# B&R Automation Studio project EFI (part 5)

### Hardware
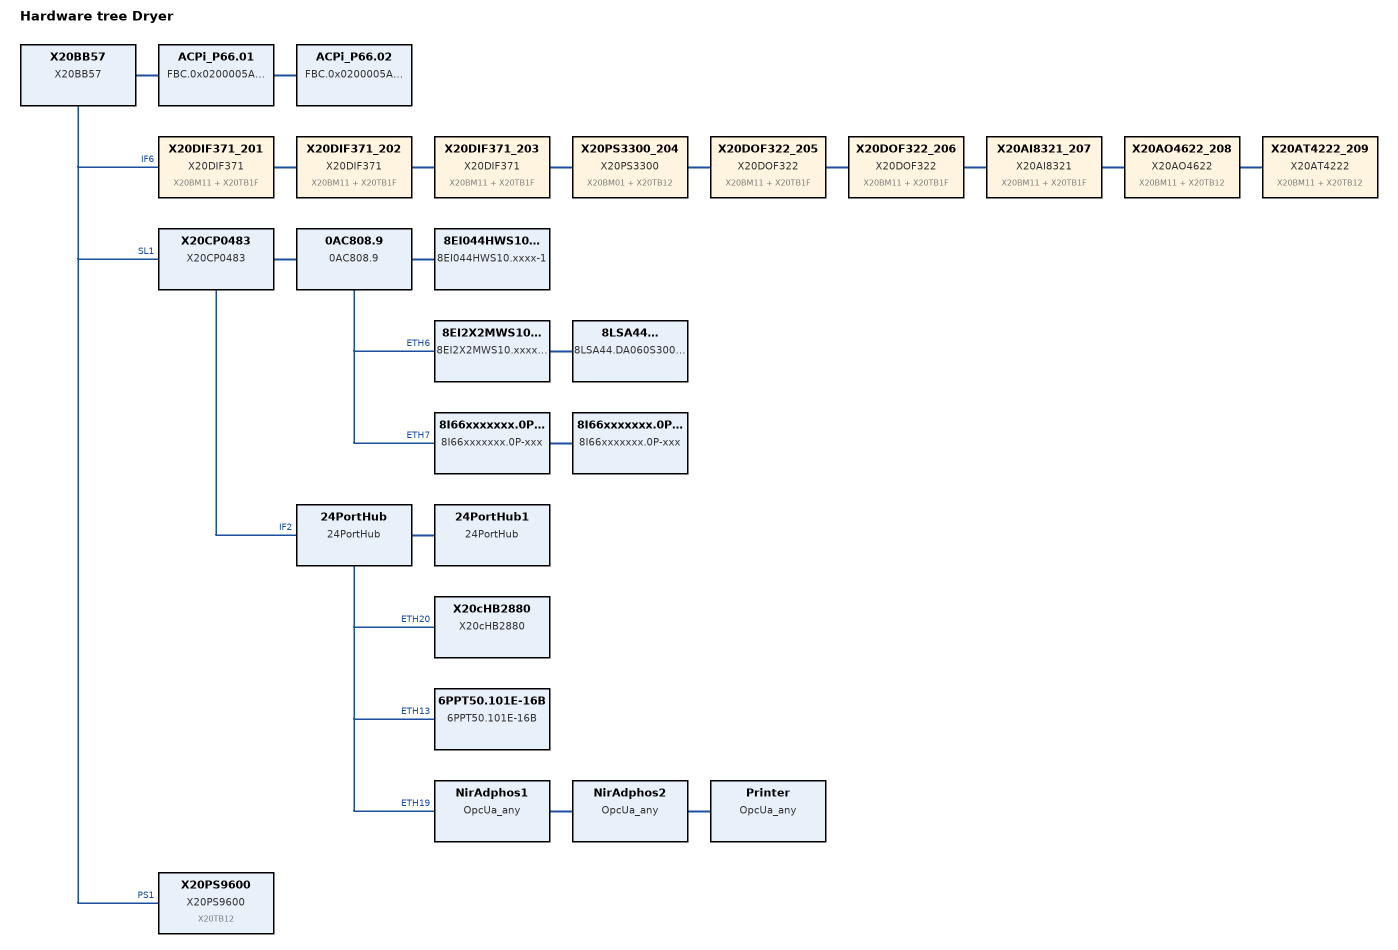
```
0AC808.9 : 0AC808.9 v1.0.0.0  [ETH1 -> X20CP0483.IF3 [Cable Type=PowerlinkCable, Length=10, Version=1.0.0.3]; ETH5 -> 8EI044HWS10.xxxx-1_BELT.PLK1 [Cable Type=PowerlinkCable, Length=10, Version=1.0.0.3]; ETH6 -> 8EI2X2MWS10.xxxx-1.PLK1 [Cable Type=PowerlinkCable, Length=10, Version=1.0.0.3]; ETH7 -> 8I66xxxxxxx.0P-81.PLK1 [Cable Type=PowerlinkCable, Length=10, Version=1.0.0.3]]
24PortHub : 24PortHub v1.0.0.1  [ETH7 -> X20CP0483.IF2 [Cable Type=PowerlinkCable, Length=10, Version=1.0.0.3]; ETH13 -> 6PPT50.101E-16B.ETH1 [Cable Type=PowerlinkCable, Length=10, Version=1.0.0.3]; ETH19 -> NirAdphos1.ETH1 [Cable Type=PowerlinkCable, Length=10, Version=1.0.0.3]; ETH20 -> X20cHB2880.ETH1 [Cable Type=PowerlinkCable, Length=10, Version=1.0.0.3]; ETH24 -> 24PortHub1.ETH3 [Cable Type=PowerlinkCable, Length=10, Version=1.0.0.3]]
24PortHub1 : 24PortHub v1.0.0.1  [ETH3 -> 24PortHub.ETH24 [Cable Type=PowerlinkCable, Length=10, Version=1.0.0.3]]
6PPT50.101E-16B : 6PPT50.101E-16B v1.3.8.0  [ETH1 -> 24PortHub.ETH13 [Cable Type=PowerlinkCable, Length=10, Version=1.0.0.3]]
  Terminal = true
  Startmode = 2
  ShowBootlogoWeb = 1
  Mode = Manual
  InternetAddress = 192.168.125.48
  Subnetmask = 255.255.255.0
  Hostname = efi_dryer_hmi
  Screensaver = 1
  Screensavertype = 0
  ActivateBuzzer = 1
  PasswordVNC = 
  SelectedFavoriteWeb = 192.168.125.47:81/index.html
  Favorites_Web1 = 
  BrowserVKeyboard = 0
  PasswordCIFS = 
  PasswordService = 
  ANSLAuthUserName = 
8EI044HWS10.xxxx-1_BELT : 8EI044HWS10.xxxx-1 v2.3.1.1  [PLK1 -> 0AC808.9.ETH5 [Cable Type=PowerlinkCable, Length=10, Version=1.0.0.3]]
  MotionTP = Acp10Arnc0
  Ax1Interface = Ax1EnDat
8EI2X2MWS10.xxxx-1 : 8EI2X2MWS10.xxxx-1 v2.3.1.1  [PLK1 -> 0AC808.9.ETH6 (NodeNumber=21) [Cable Type=PowerlinkCable, Length=10, Version=1.0.0.3]; EC1 -> 8LSA44.DA060S300-3.EC]
  MotionTP = Acp10Arnc0
  Ax1Interface = Ax1EnDat
8I66xxxxxxx.0P-81 : 8I66xxxxxxx.0P-xxx v2.5.1.0  [PLK1 -> 0AC808.9.ETH7 (NodeNumber=81) [Cable Type=PowerlinkCable, Length=10, Version=1.0.0.3]; PLK2 -> 8I66xxxxxxx.0P-82.PLK1 (NodeNumber=81) [Cable Type=PowerlinkCable, Length=10, Version=1.0.0.3]]
  FunctionModel = Standard
  Supervision = off
  UnitOfSetpoint = Rpm
  IOM_AIDP1 = LFT
  IOM_AIDP2 = LCR
  IOM_AIDP3 = OTRN
  IOM_AIDP4 = IL1R
  IOM_AIDP5 = AI1R
  IOM_AIDP6 = AI2R
  IOM_AIDP7 = AI3R
  IOM_AIDP8 = OL1I
  IOM_AIDP9 = AO1I
  IOM_R1ctrl = mapped
  IOM_R2ctrl = mapped
  IOM_LO1ctrl = mapped
  IOM_AO1ctrl = mapped
  Sel_AO1T = 0A
  Sel_NameplateMask = 8Ix6T401500_IEC
  Cfg_NSP = 2940
  Cfg_NCR = 277
  Cfg_COS = 82
  Sel_TUN = AUTO
8I66xxxxxxx.0P-82 : 8I66xxxxxxx.0P-xxx v2.5.1.0  [PLK1 -> 8I66xxxxxxx.0P-81.PLK2 [Cable Type=PowerlinkCable, Length=10, Version=1.0.0.3]]
  FunctionModel = Standard
  Supervision = off
  UnitOfSetpoint = Rpm
  IOM_AIDP1 = LFT
  IOM_AIDP2 = LCR
  IOM_AIDP3 = OTRN
  IOM_AIDP4 = IL1R
  IOM_AIDP5 = AI1R
  IOM_AIDP6 = AI2R
  IOM_AIDP7 = AI3R
  IOM_AIDP8 = OL1I
  IOM_AIDP9 = AO1I
  IOM_R1ctrl = mapped
  IOM_R2ctrl = mapped
  IOM_LO1ctrl = mapped
  IOM_AO1ctrl = mapped
  Sel_AO1T = 0A
  Sel_NameplateMask = 8Ix6T401500_IEC
  Cfg_NSP = 2940
  Cfg_NCR = 277
  Cfg_COS = 82
  Sel_TUN = AUTO
8LSA44.DA060S300-3 : 8LSA44.DA060S300-3 v1.0.10.37  [EC -> 8EI2X2MWS10.xxxx-1.EC1; MT -> 8EI2X2MWS10.xxxx-1.MT1]
ACPi_P66.01 : FBC.0x0200005A.320.ACPi_P66_P76 v1.3 (OrderNumber=ACPi_P66_P76)  [CAN1 -> X20BB57.IF7 (NodeNumber=81)]
  p2002sub5_connecttomaster = 2
  p2016sub3_connecttomaster = 1
  p2016subd_connecttomaster = 5
  p2016sub21_connecttomaster = 1
  p2016sub22_connecttomaster = 1
  p2016sub3e_connecttomaster = 5
  p2029sub16_connecttomaster = 2
  p2038sub2_connecttomaster = 4
  p2038sub3_connecttomaster = 4
  p2038sub4_connecttomaster = 2
  p2038sub5_connecttomaster = 2
  p203csub2_connecttomaster = 5
  p203csub3_connecttomaster = 5
  p6040_connecttomaster = 0
  p6041_connecttomaster = 0
  p6042_connecttomaster = 0
  p6044_connecttomaster = 0
  p6077_connecttomaster = 1
  p1800_transmissionselection = 2
  p1801_transmissionselection = 2
  p1802_transmissionselection = 2
ACPi_P66.02 : FBC.0x0200005A.320.ACPi_P66_P76 v1.3 (OrderNumber=ACPi_P66_P76)  [CAN1 -> ACPi_P66.01.CAN2]
  p2002sub5_connecttomaster = 2
  p2016sub3_connecttomaster = 1
  p2016subd_connecttomaster = 5
  p2016sub21_connecttomaster = 1
  p2016sub22_connecttomaster = 1
  p2016sub3e_connecttomaster = 5
  p2029sub16_connecttomaster = 2
  p2038sub2_connecttomaster = 4
  p2038sub3_connecttomaster = 4
  p2038sub4_connecttomaster = 2
  p2038sub5_connecttomaster = 2
  p203csub2_connecttomaster = 5
  p203csub3_connecttomaster = 5
  p6040_connecttomaster = 0
  p6041_connecttomaster = 0
  p6042_connecttomaster = 0
  p6044_connecttomaster = 0
  p6077_connecttomaster = 1
  p1800_transmissionselection = 2
  p1801_transmissionselection = 2
  p1802_transmissionselection = 2
NirAdphos1 : OpcUa_any v1.0.0.1  [ETH1 -> 24PortHub.ETH19 [Cable Type=PowerlinkCable, Length=10, Version=1.0.0.3]; ETH2 -> NirAdphos2.ETH1 [Cable Type=PowerlinkCable, Length=10, Version=1.0.0.3]]
  ServerDiagnostics = on
  ServerEndpointUrl = opc.tcp://192.168.125.91:4840
  PnPTimeout = 2500
  SecurityMsgMode = 0
  Channel1
  ChannelID1 = HMI
  ChannelBrowsePath1 = /0:Root/0:Objects/3:ServerInterfaces/4:SendData/4:DB11_HMI_out/4:HMI
  ChannelType1 = INT
  Channel2
  ChannelID2 = Hardware
  ChannelBrowsePath2 = /0:Root/0:Objects/3:ServerInterfaces/4:SendData/4:DB11_HMI_out/4:Hardware
  ChannelType2 = INT
  Channel3
  ChannelID3 = Software
  ChannelBrowsePath3 = /0:Root/0:Objects/3:ServerInterfaces/4:SendData/4:DB11_HMI_out/4:Software
  ChannelType3 = INT
  Channel4
  ChannelID4 = Interface
  ChannelBrowsePath4 = /0:Root/0:Objects/3:ServerInterfaces/4:SendData/4:DB11_HMI_out/4:interface
  ChannelType4 = INT
  Channel5
  ChannelID5 = NIRno
  ChannelBrowsePath5 = /0:Root/0:Objects/3:ServerInterfaces/4:SendData/4:DB11_HMI_out/4:general/4:NIRno
  ChannelType5 = INT
  Channel6
  ChannelID6 = NIRwidth
  ChannelBrowsePath6 = /0:Root/0:Objects/3:ServerInterfaces/4:SendData/4:DB11_HMI_out/4:general/4:NIRwidth
  ChannelType6 = INT
  Channel7
  ChannelID7 = calPower
  ChannelBrowsePath7 = /0:Root/0:Objects/3:ServerInterfaces/4:SendData/4:DB11_HMI_out/4:general/4:calPower
  ChannelType7 = INT
  Channel8
  ChannelID8 = speed
  ChannelBrowsePath8 = /0:Root/0:Objects/3:ServerInterfaces/4:SendData/4:DB11_HMI_out/4:general/4:speed
  ChannelType8 = REAL
  Channel9
  ChannelID9 = Watchdog1
  ChannelBrowsePath9 = /0:Root/0:Objects/3:ServerInterfaces/4:SendData/4:DB11_HMI_out/4:general/4:Watchdog
  Channel10
  ChannelID10 = EmFailNo_1
  ChannelBrowsePath10 = /0:Root/0:Objects/3:ServerInterfaces/4:SendData/4:DB11_HMI_out/4:module/4:[1]/4:EmFailNo
  ChannelType10 = USINT
  Channel11
  ChannelID11 = EmFailNo_2
  ChannelBrowsePath11 = /0:Root/0:Objects/3:ServerInterfaces/4:SendData/4:DB11_HMI_out/4:module/4:[2]/4:EmFailNo
  ChannelType11 = USINT
  Channel12
  ChannelID12 = ExhAirRunning_1
  ChannelBrowsePath12 = /0:Root/0:Objects/3:ServerInterfaces/4:SendData/4:DB11_HMI_out/4:module/4:[1]/4:ExhAirRunning
  Channel13
  ChannelID13 = ExhAirRunning_2
  ChannelBrowsePath13 = /0:Root/0:Objects/3:ServerInterfaces/4:SendData/4:DB11_HMI_out/4:module/4:[2]/4:ExhAirRunning
  Channel14
  ChannelID14 = NIRstatus_1
  ChannelBrowsePath14 = /0:Root/0:Objects/3:ServerInterfaces/4:SendData/4:DB11_HMI_out/4:module/4:[1]/4:NIRstatus
  ChannelType14 = INT
  Channel15
  ChannelID15 = NIRstatus_2
  ChannelBrowsePath15 = /0:Root/0:Objects/3:ServerInterfaces/4:SendData/4:DB11_HMI_out/4:module/4:[2]/4:NIRstatus
  ChannelType15 = INT
  Channel16
  ChannelID16 = airPressIn_1
  ChannelBrowsePath16 = /0:Root/0:Objects/3:ServerInterfaces/4:SendData/4:DB11_HMI_out/4:module/4:[1]/4:airPressIn
  ChannelType16 = REAL
  Channel17
  ChannelID17 = airPressIn_2
  ChannelBrowsePath17 = /0:Root/0:Objects/3:ServerInterfaces/4:SendData/4:DB11_HMI_out/4:module/4:[2]/4:airPressIn
  ChannelType17 = REAL
  Channel18
  ChannelID18 = airPressOut_1
  ChannelBrowsePath18 = /0:Root/0:Objects/3:ServerInterfaces/4:SendData/4:DB11_HMI_out/4:module/4:[1]/4:airPressOut
  ChannelType18 = REAL
  Channel19
  ChannelID19 = airPressOut_2
  ChannelBrowsePath19 = /0:Root/0:Objects/3:ServerInterfaces/4:SendData/4:DB11_HMI_out/4:module/4:[2]/4:airPressOut
  ChannelType19 = REAL
  Channel20
  ChannelID20 = airFilter_1
  ChannelBrowsePath20 = /0:Root/0:Objects/3:ServerInterfaces/4:SendData/4:DB11_HMI_out/4:module/4:[1]/4:airFilter
  ChannelType20 = INT
  Channel21
  ChannelID21 = airFilter_2
  ChannelBrowsePath21 = /0:Root/0:Objects/3:ServerInterfaces/4:SendData/4:DB11_HMI_out/4:module/4:[2]/4:airFilter
  ChannelType21 = INT
  Channel22
  ChannelID22 = actSpeedIn_1
  ChannelBrowsePath22 = /0:Root/0:Objects/3:ServerInterfaces/4:SendData/4:DB11_HMI_out/4:module/4:[1]/4:actSpeedIn
  ChannelType22 = INT
  Channel23
  ChannelID23 = actSpeedIn_2
  ChannelBrowsePath23 = /0:Root/0:Objects/3:ServerInterfaces/4:SendData/4:DB11_HMI_out/4:module/4:[2]/4:actSpeedIn
  ChannelType23 = INT
  Channel24
  ChannelID24 = actSpeedOut_1
  ChannelBrowsePath24 = /0:Root/0:Objects/3:ServerInterfaces/4:SendData/4:DB11_HMI_out/4:module/4:[1]/4:actSpeedOut
  ChannelType24 = INT
  Channel25
  ChannelID25 = actSpeedOut_2
  ChannelBrowsePath25 = /0:Root/0:Objects/3:ServerInterfaces/4:SendData/4:DB11_HMI_out/4:module/4:[2]/4:actSpeedOut
  ChannelType25 = INT
  Channel26
  ChannelID26 = actPower_1
  ChannelBrowsePath26 = /0:Root/0:Objects/3:ServerInterfaces/4:SendData/4:DB11_HMI_out/4:module/4:[1]/4:actPower
  ChannelType26 = INT
  Channel27
  ChannelID27 = actPower_2
  ChannelBrowsePath27 = /0:Root/0:Objects/3:ServerInterfaces/4:SendData/4:DB11_HMI_out/4:module/4:[2]/4:actPower
  ChannelType27 = INT
  Channel28
  ChannelID28 = Watchdog2
  ChannelBrowsePath28 = /0:Root/0:Objects/3:ServerInterfaces/4:SendData/4:DB11_HMI_out/4:general/4:Watchdog
  Channel29
  ChannelID29 = Reset
  ChannelBrowsePath29 = /0:Root/0:Objects/3:ServerInterfaces/5:RecData/5:DB10_HMI_in/5:reset
  ChannelDirection29 = OUT
  Channel30
  ChannelID30 = Pend
  ChannelBrowsePath30 = /0:Root/0:Objects/3:ServerInterfaces/5:RecData/5:DB10_HMI_in/5:product/5:Pend
  ChannelDirection30 = OUT
  ChannelType30 = REAL
  Channel31
  ChannelID31 = Pstart
  ChannelBrowsePath31 = /0:Root/0:Objects/3:ServerInterfaces/5:RecData/5:DB10_HMI_in/5:product/5:Pstart
  ChannelDirection31 = OUT
  ChannelType31 = REAL
  Channel32
  ChannelID32 = Vend
  ChannelBrowsePath32 = /0:Root/0:Objects/3:ServerInterfaces/5:RecData/5:DB10_HMI_in/5:product/5:Vend
  ChannelDirection32 = OUT
  ChannelType32 = REAL
  Channel33
  ChannelID33 = Vstart
  ChannelBrowsePath33 = /0:Root/0:Objects/3:ServerInterfaces/5:RecData/5:DB10_HMI_in/5:product/5:Vstart
  ChannelDirection33 = OUT
  ChannelType33 = REAL
  Channel34
  ChannelID34 = AdjPos
  ChannelBrowsePath34 = /0:Root/0:Objects/3:ServerInterfaces/5:RecData/5:DB10_HMI_in/5:product/5:adjPos
  ChannelDirection34 = OUT
  ChannelType34 = INT
  Channel35
  ChannelID35 = WebWidth
  ChannelBrowsePath35 = /0:Root/0:Objects/3:ServerInterfaces/5:RecData/5:DB10_HMI_in/5:product/5:webWidth
  ChannelDirection35 = OUT
  ChannelType35 = INT
  Channel36
  ChannelID36 = Adjust_1
  ChannelBrowsePath36 = /0:Root/0:Objects/3:ServerInterfaces/5:RecData/5:DB10_HMI_in/5:module/5:[1]/5:adjust
  ChannelDirection36 = OUT
  ChannelType36 = INT
  Channel37
  ChannelID37 = Adjust_2
  ChannelBrowsePath37 = /0:Root/0:Objects/3:ServerInterfaces/5:RecData/5:DB10_HMI_in/5:module/5:[2]/5:adjust
  ChannelDirection37 = OUT
  ChannelType37 = INT
  Channel38
  ChannelID38 = EnableMod_1
  ChannelBrowsePath38 = /0:Root/0:Objects/3:ServerInterfaces/5:RecData/5:DB10_HMI_in/5:module/5:[1]/5:enableMod
  ChannelDirection38 = OUT
  Channel39
  ChannelID39 = EnableMod_2
  ChannelBrowsePath39 = /0:Root/0:Objects/3:ServerInterfaces/5:RecData/5:DB10_HMI_in/5:module/5:[2]/5:enableMod
  ChannelDirection39 = OUT
  Channel40
  ChannelID40 = WatchdogOut
  ChannelBrowsePath40 = /0:Root/0:Objects/3:ServerInterfaces/5:RecData/5:DB10_HMI_in/5:Watchdog
  ChannelDirection40 = OUT
  Channel41
  ChannelID41 = Enable_DDC
  ChannelBrowsePath41 = /0:Root/0:Objects/3:ServerInterfaces/5:RecData/5:DB10_HMI_in/5:DDCon
  ChannelDirection41 = OUT
  Channel42
  ChannelID42 = NIR1_Int1
  ChannelBrowsePath42 = /0:Root/0:Objects/3:ServerInterfaces/5:RecData/5:DB10_HMI_in/5:intensity/5:intensity/5:[1]
  ChannelDirection42 = OUT
  ChannelType42 = INT
  Channel43
  ChannelID43 = NIR1_Int2
  ChannelBrowsePath43 = /0:Root/0:Objects/3:ServerInterfaces/5:RecData/5:DB10_HMI_in/5:intensity/5:intensity/5:[2]
  ChannelDirection43 = OUT
  ChannelType43 = INT
  Channel44
  ChannelID44 = NIR1_Int3
  ChannelBrowsePath44 = /0:Root/0:Objects/3:ServerInterfaces/5:RecData/5:DB10_HMI_in/5:intensity/5:intensity/5:[3]
  ChannelDirection44 = OUT
  ChannelType44 = INT
  Channel45
  ChannelID45 = NIR1_Int4
  ChannelBrowsePath45 = /0:Root/0:Objects/3:ServerInterfaces/5:RecData/5:DB10_HMI_in/5:intensity/5:intensity/5:[4]
  ChannelDirection45 = OUT
  ChannelType45 = INT
  Channel46
  ChannelID46 = NIR1_Int5
  ChannelBrowsePath46 = /0:Root/0:Objects/3:ServerInterfaces/5:RecData/5:DB10_HMI_in/5:intensity/5:intensity/5:[5]
  ChannelDirection46 = OUT
  ChannelType46 = INT
  Channel47
  ChannelID47 = NIR1_Int6
  ChannelBrowsePath47 = /0:Root/0:Objects/3:ServerInterfaces/5:RecData/5:DB10_HMI_in/5:intensity/5:intensity/5:[6]
  ChannelDirection47 = OUT
  ChannelType47 = INT
  Channel48
  ChannelID48 = NIR1_Int7
  ChannelBrowsePath48 = /0:Root/0:Objects/3:ServerInterfaces/5:RecData/5:DB10_HMI_in/5:intensity/5:intensity/5:[7]
  ChannelDirection48 = OUT
  ChannelType48 = INT
  Channel49
  ChannelID49 = NIR1_Int8
  ChannelBrowsePath49 = /0:Root/0:Objects/3:ServerInterfaces/5:RecData/5:DB10_HMI_in/5:intensity/5:intensity/5:[8]
  ChannelDirection49 = OUT
  ChannelType49 = INT
  Channel50
  ChannelID50 = NIR1_Int9
  ChannelBrowsePath50 = /0:Root/0:Objects/3:ServerInterfaces/5:RecData/5:DB10_HMI_in/5:intensity/5:intensity/5:[9]
  ChannelDirection50 = OUT
  ChannelType50 = INT
  Channel51
  ChannelID51 = NIR1_Int10
  ChannelBrowsePath51 = /0:Root/0:Objects/3:ServerInterfaces/5:RecData/5:DB10_HMI_in/5:intensity/5:intensity/5:[10]
  ChannelDirection51 = OUT
  ChannelType51 = INT
  Channel52
  ChannelID52 = NIR1_Int11
  ChannelBrowsePath52 = /0:Root/0:Objects/3:ServerInterfaces/5:RecData/5:DB10_HMI_in/5:intensity/5:intensity/5:[11]
  ChannelDirection52 = OUT
  ChannelType52 = INT
  Channel53
  ChannelID53 = NIR1_Int12
  ChannelBrowsePath53 = /0:Root/0:Objects/3:ServerInterfaces/5:RecData/5:DB10_HMI_in/5:intensity/5:intensity/5:[12]
  ChannelDirection53 = OUT
  ChannelType53 = INT
  Channel54
  ChannelID54 = NIR1_Int13
  ChannelBrowsePath54 = /0:Root/0:Objects/3:ServerInterfaces/5:RecData/5:DB10_HMI_in/5:intensity/5:intensity/5:[13]
  ChannelDirection54 = OUT
  ChannelType54 = INT
  Channel55
  ChannelID55 = NIR1_Int14
  ChannelBrowsePath55 = /0:Root/0:Objects/3:ServerInterfaces/5:RecData/5:DB10_HMI_in/5:intensity/5:intensity/5:[14]
  ChannelDirection55 = OUT
  ChannelType55 = INT
  Channel56
  ChannelID56 = NIR1_Int15
  ChannelBrowsePath56 = /0:Root/0:Objects/3:ServerInterfaces/5:RecData/5:DB10_HMI_in/5:intensity/5:intensity/5:[15]
  ChannelDirection56 = OUT
  ChannelType56 = INT
  Channel57
  ChannelID57 = NIR1_Int16
  ChannelBrowsePath57 = /0:Root/0:Objects/3:ServerInterfaces/5:RecData/5:DB10_HMI_in/5:intensity/5:intensity/5:[16]
  ChannelDirection57 = OUT
  ChannelType57 = INT
  Channel58
  ChannelID58 = NIR1_Int17
  ChannelBrowsePath58 = /0:Root/0:Objects/3:ServerInterfaces/5:RecData/5:DB10_HMI_in/5:intensity/5:intensity/5:[17]
  ChannelDirection58 = OUT
  ChannelType58 = INT
  Channel59
  ChannelID59 = NIR1_Int18
  ChannelBrowsePath59 = /0:Root/0:Objects/3:ServerInterfaces/5:RecData/5:DB10_HMI_in/5:intensity/5:intensity/5:[18]
  ChannelDirection59 = OUT
  ChannelType59 = INT
  Channel60
  ChannelID60 = NIR1_Int19
  ChannelBrowsePath60 = /0:Root/0:Objects/3:ServerInterfaces/5:RecData/5:DB10_HMI_in/5:intensity/5:intensity/5:[19]
  ChannelDirection60 = OUT
  ChannelType60 = INT
  Channel61
  ChannelID61 = NIR1_Int20
  ChannelBrowsePath61 = /0:Root/0:Objects/3:ServerInterfaces/5:RecData/5:DB10_HMI_in/5:intensity/5:intensity/5:[20]
  ChannelDirection61 = OUT
  ChannelType61 = INT
  Channel62
  ChannelID62 = NIR1_Int21
  ChannelBrowsePath62 = /0:Root/0:Objects/3:ServerInterfaces/5:RecData/5:DB10_HMI_in/5:intensity/5:intensity/5:[21]
  ChannelDirection62 = OUT
  ChannelType62 = INT
  Channel63
  ChannelID63 = NIR1_Int22
  ChannelBrowsePath63 = /0:Root/0:Objects/3:ServerInterfaces/5:RecData/5:DB10_HMI_in/5:intensity/5:intensity/5:[22]
  ChannelDirection63 = OUT
  ChannelType63 = INT
  Channel64
  ChannelID64 = NIR1_Int23
  ChannelBrowsePath64 = /0:Root/0:Objects/3:ServerInterfaces/5:RecData/5:DB10_HMI_in/5:intensity/5:intensity/5:[23]
  ChannelDirection64 = OUT
  ChannelType64 = INT
  Channel65
  ChannelID65 = NIR1_Int24
  ChannelBrowsePath65 = /0:Root/0:Objects/3:ServerInterfaces/5:RecData/5:DB10_HMI_in/5:intensity/5:intensity/5:[24]
  ChannelDirection65 = OUT
  ChannelType65 = INT
  Channel66
  ChannelID66 = NIR1_Int25
  ChannelBrowsePath66 = /0:Root/0:Objects/3:ServerInterfaces/5:RecData/5:DB10_HMI_in/5:intensity/5:intensity/5:[25]
  ChannelDirection66 = OUT
  ChannelType66 = INT
  Channel67
  ChannelID67 = NIR1_Int26
  ChannelBrowsePath67 = /0:Root/0:Objects/3:ServerInterfaces/5:RecData/5:DB10_HMI_in/5:intensity/5:intensity/5:[26]
  ChannelDirection67 = OUT
  ChannelType67 = INT
  Channel68
  ChannelID68 = NIR1_Int27
  ChannelBrowsePath68 = /0:Root/0:Objects/3:ServerInterfaces/5:RecData/5:DB10_HMI_in/5:intensity/5:intensity/5:[27]
  ChannelDirection68 = OUT
  ChannelType68 = INT
  Channel69
  ChannelID69 = NIR1_Int28
  ChannelBrowsePath69 = /0:Root/0:Objects/3:ServerInterfaces/5:RecData/5:DB10_HMI_in/5:intensity/5:intensity/5:[28]
  ChannelDirection69 = OUT
  ChannelType69 = INT
  Channel70
  ChannelID70 = NIR1_Int29
  ChannelBrowsePath70 = /0:Root/0:Objects/3:ServerInterfaces/5:RecData/5:DB10_HMI_in/5:intensity/5:intensity/5:[29]
  ChannelDirection70 = OUT
  ChannelType70 = INT
  Channel71
  ChannelID71 = NIR1_Int30
  ChannelBrowsePath71 = /0:Root/0:Objects/3:ServerInterfaces/5:RecData/5:DB10_HMI_in/5:intensity/5:intensity/5:[30]
  ChannelDirection71 = OUT
  ChannelType71 = INT
  Channel72
  ChannelID72 = NIR1_Int31
  ChannelBrowsePath72 = /0:Root/0:Objects/3:ServerInterfaces/5:RecData/5:DB10_HMI_in/5:intensity/5:intensity/5:[31]
  ChannelDirection72 = OUT
  ChannelType72 = INT
  Channel73
  ChannelID73 = NIR1_Int32
  ChannelBrowsePath73 = /0:Root/0:Objects/3:ServerInterfaces/5:RecData/5:DB10_HMI_in/5:intensity/5:intensity/5:[32]
  ChannelDirection73 = OUT
  ChannelType73 = INT
  Channel74
  ChannelID74 = NIR1_Int33
  ChannelBrowsePath74 = /0:Root/0:Objects/3:ServerInterfaces/5:RecData/5:DB10_HMI_in/5:intensity/5:intensity/5:[33]
  ChannelDirection74 = OUT
  ChannelType74 = INT
  Channel75
  ChannelID75 = NIR1_Int34
  ChannelBrowsePath75 = /0:Root/0:Objects/3:ServerInterfaces/5:RecData/5:DB10_HMI_in/5:intensity/5:intensity/5:[34]
  ChannelDirection75 = OUT
  ChannelType75 = INT
  Channel76
  ChannelID76 = NIR1_Int35
  ChannelBrowsePath76 = /0:Root/0:Objects/3:ServerInterfaces/5:RecData/5:DB10_HMI_in/5:intensity/5:intensity/5:[35]
  ChannelDirection76 = OUT
  ChannelType76 = INT
  Channel77
  ChannelID77 = NIR1_Int36
  ChannelBrowsePath77 = /0:Root/0:Objects/3:ServerInterfaces/5:RecData/5:DB10_HMI_in/5:intensity/5:intensity/5:[36]
  ChannelDirection77 = OUT
  ChannelType77 = INT
  Channel78
  ChannelID78 = NIR1_Int37
  ChannelBrowsePath78 = /0:Root/0:Objects/3:ServerInterfaces/5:RecData/5:DB10_HMI_in/5:intensity/5:intensity/5:[37]
  ChannelDirection78 = OUT
  ChannelType78 = INT
  Channel79
  ChannelID79 = NIR1_Int38
  ChannelBrowsePath79 = /0:Root/0:Objects/3:ServerInterfaces/5:RecData/5:DB10_HMI_in/5:intensity/5:intensity/5:[38]
  ChannelDirection79 = OUT
  ChannelType79 = INT
  Channel80
  ChannelID80 = NIR1_Int39
  ChannelBrowsePath80 = /0:Root/0:Objects/3:ServerInterfaces/5:RecData/5:DB10_HMI_in/5:intensity/5:intensity/5:[39]
  ChannelDirection80 = OUT
  ChannelType80 = INT
  Channel81
  ChannelID81 = NIR1_Int40
  ChannelBrowsePath81 = /0:Root/0:Objects/3:ServerInterfaces/5:RecData/5:DB10_HMI_in/5:intensity/5:intensity/5:[40]
  ChannelDirection81 = OUT
  ChannelType81 = INT
  Channel82
  ChannelID82 = NIR1_Int41
  ChannelBrowsePath82 = /0:Root/0:Objects/3:ServerInterfaces/5:RecData/5:DB10_HMI_in/5:intensity/5:intensity/5:[41]
  ChannelDirection82 = OUT
  ChannelType82 = INT
  Channel83
  ChannelID83 = NIR1_Int42
  ChannelBrowsePath83 = /0:Root/0:Objects/3:ServerInterfaces/5:RecData/5:DB10_HMI_in/5:intensity/5:intensity/5:[42]
  ChannelDirection83 = OUT
  ChannelType83 = INT
  Channel84
  ChannelID84 = NIR1_Int43
  ChannelBrowsePath84 = /0:Root/0:Objects/3:ServerInterfaces/5:RecData/5:DB10_HMI_in/5:intensity/5:intensity/5:[43]
  ChannelDirection84 = OUT
  ChannelType84 = INT
  Channel85
  ChannelID85 = NIR1_Int44
  ChannelBrowsePath85 = /0:Root/0:Objects/3:ServerInterfaces/5:RecData/5:DB10_HMI_in/5:intensity/5:intensity/5:[44]
  ChannelDirection85 = OUT
  ChannelType85 = INT
  Channel86
  ChannelID86 = NIR1_Int45
  ChannelBrowsePath86 = /0:Root/0:Objects/3:ServerInterfaces/5:RecData/5:DB10_HMI_in/5:intensity/5:intensity/5:[45]
  ChannelDirection86 = OUT
  ChannelType86 = INT
  Channel87
  ChannelID87 = NIR1_Int46
  ChannelBrowsePath87 = /0:Root/0:Objects/3:ServerInterfaces/5:RecData/5:DB10_HMI_in/5:intensity/5:intensity/5:[46]
  ChannelDirection87 = OUT
  ChannelType87 = INT
  Channel88
  ChannelID88 = NIR1_Int47
  ChannelBrowsePath88 = /0:Root/0:Objects/3:ServerInterfaces/5:RecData/5:DB10_HMI_in/5:intensity/5:intensity/5:[47]
  ChannelDirection88 = OUT
  ChannelType88 = INT
  Channel89
  ChannelID89 = NIR1_Int48
  ChannelBrowsePath89 = /0:Root/0:Objects/3:ServerInterfaces/5:RecData/5:DB10_HMI_in/5:intensity/5:intensity/5:[48]
  ChannelDirection89 = OUT
  ChannelType89 = INT
NirAdphos2 : OpcUa_any v1.0.0.1  [ETH1 -> NirAdphos1.ETH2 [Cable Type=PowerlinkCable, Length=10, Version=1.0.0.3]; ETH2 -> Printer.ETH1 [Cable Type=PowerlinkCable, Length=10, Version=1.0.0.3]]
  ServerDiagnostics = on
  ServerEndpointUrl = opc.tcp://192.168.125.92:4840
  PnPTimeout = 2500
  SecurityMsgMode = 0
  Channel1
  ChannelID1 = NIR2_Int1
  ChannelBrowsePath1 = /0:Root/0:Objects/3:ServerInterfaces/0:RecData/4:DB10_HMI_in/4:intensity/4:[1]
  ChannelDirection1 = OUT
  ChannelType1 = INT
  Channel2
  ChannelID2 = NIR2_Int2
  ChannelBrowsePath2 = /0:Root/0:Objects/3:ServerInterfaces/0:RecData/4:DB10_HMI_in/4:intensity/4:[2]
  ChannelDirection2 = OUT
  ChannelType2 = INT
  Channel3
  ChannelID3 = NIR2_Int3
  ChannelBrowsePath3 = /0:Root/0:Objects/3:ServerInterfaces/0:RecData/4:DB10_HMI_in/4:intensity/4:[3]
  ChannelDirection3 = OUT
  ChannelType3 = INT
  Channel4
  ChannelID4 = NIR2_Int4
  ChannelBrowsePath4 = /0:Root/0:Objects/3:ServerInterfaces/0:RecData/4:DB10_HMI_in/4:intensity/4:[4]
  ChannelDirection4 = OUT
  ChannelType4 = INT
  Channel5
  ChannelID5 = NIR2_Int5
  ChannelBrowsePath5 = /0:Root/0:Objects/3:ServerInterfaces/0:RecData/4:DB10_HMI_in/4:intensity/4:[5]
  ChannelDirection5 = OUT
  ChannelType5 = INT
  Channel6
  ChannelID6 = NIR2_Int6
  ChannelBrowsePath6 = /0:Root/0:Objects/3:ServerInterfaces/0:RecData/4:DB10_HMI_in/4:intensity/4:[6]
  ChannelDirection6 = OUT
  ChannelType6 = INT
  Channel7
  ChannelID7 = NIR2_Int7
  ChannelBrowsePath7 = /0:Root/0:Objects/3:ServerInterfaces/0:RecData/4:DB10_HMI_in/4:intensity/4:[7]
  ChannelDirection7 = OUT
  ChannelType7 = INT
  Channel8
  ChannelID8 = NIR2_Int8
  ChannelBrowsePath8 = /0:Root/0:Objects/3:ServerInterfaces/0:RecData/4:DB10_HMI_in/4:intensity/4:[8]
  ChannelDirection8 = OUT
  ChannelType8 = INT
  Channel9
  ChannelID9 = NIR2_Int9
  ChannelBrowsePath9 = /0:Root/0:Objects/3:ServerInterfaces/0:RecData/4:DB10_HMI_in/4:intensity/4:[9]
  ChannelDirection9 = OUT
  ChannelType9 = INT
  Channel10
  ChannelID10 = NIR2_Int10
  ChannelBrowsePath10 = /0:Root/0:Objects/3:ServerInterfaces/0:RecData/4:DB10_HMI_in/4:intensity/4:[10]
  ChannelDirection10 = OUT
  ChannelType10 = INT
  Channel11
  ChannelID11 = NIR2_Int11
  ChannelBrowsePath11 = /0:Root/0:Objects/3:ServerInterfaces/0:RecData/4:DB10_HMI_in/4:intensity/4:[11]
  ChannelDirection11 = OUT
  ChannelType11 = INT
  Channel12
  ChannelID12 = NIR2_Int12
  ChannelBrowsePath12 = /0:Root/0:Objects/3:ServerInterfaces/0:RecData/4:DB10_HMI_in/4:intensity/4:[12]
  ChannelDirection12 = OUT
  ChannelType12 = INT
  Channel13
  ChannelID13 = NIR2_Int13
  ChannelBrowsePath13 = /0:Root/0:Objects/3:ServerInterfaces/0:RecData/4:DB10_HMI_in/4:intensity/4:[13]
  ChannelDirection13 = OUT
  ChannelType13 = INT
  Channel14
  ChannelID14 = NIR2_Int14
  ChannelBrowsePath14 = /0:Root/0:Objects/3:ServerInterfaces/0:RecData/4:DB10_HMI_in/4:intensity/4:[14]
  ChannelDirection14 = OUT
  ChannelType14 = INT
  Channel15
  ChannelID15 = NIR2_Int15
  ChannelBrowsePath15 = /0:Root/0:Objects/3:ServerInterfaces/0:RecData/4:DB10_HMI_in/4:intensity/4:[15]
  ChannelDirection15 = OUT
  ChannelType15 = INT
  Channel16
  ChannelID16 = NIR2_Int16
  ChannelBrowsePath16 = /0:Root/0:Objects/3:ServerInterfaces/0:RecData/4:DB10_HMI_in/4:intensity/4:[16]
  ChannelDirection16 = OUT
  ChannelType16 = INT
  Channel17
  ChannelID17 = NIR2_Int17
  ChannelBrowsePath17 = /0:Root/0:Objects/3:ServerInterfaces/0:RecData/4:DB10_HMI_in/4:intensity/4:[17]
  ChannelDirection17 = OUT
  ChannelType17 = INT
  Channel18
  ChannelID18 = NIR2_Int18
  ChannelBrowsePath18 = /0:Root/0:Objects/3:ServerInterfaces/0:RecData/4:DB10_HMI_in/4:intensity/4:[18]
  ChannelDirection18 = OUT
  ChannelType18 = INT
  Channel19
  ChannelID19 = NIR2_Int19
  ChannelBrowsePath19 = /0:Root/0:Objects/3:ServerInterfaces/0:RecData/4:DB10_HMI_in/4:intensity/4:[19]
  ChannelDirection19 = OUT
  ChannelType19 = INT
  Channel20
  ChannelID20 = NIR2_Int20
  ChannelBrowsePath20 = /0:Root/0:Objects/3:ServerInterfaces/0:RecData/4:DB10_HMI_in/4:intensity/4:[20]
  ChannelDirection20 = OUT
  ChannelType20 = INT
  Channel21
  ChannelID21 = NIR2_Int21
  ChannelBrowsePath21 = /0:Root/0:Objects/3:ServerInterfaces/0:RecData/4:DB10_HMI_in/4:intensity/4:[21]
  ChannelDirection21 = OUT
  ChannelType21 = INT
  Channel22
  ChannelID22 = NIR2_Int22
  ChannelBrowsePath22 = /0:Root/0:Objects/3:ServerInterfaces/0:RecData/4:DB10_HMI_in/4:intensity/4:[22]
  ChannelDirection22 = OUT
  ChannelType22 = INT
  Channel23
  ChannelID23 = NIR2_Int23
  ChannelBrowsePath23 = /0:Root/0:Objects/3:ServerInterfaces/0:RecData/4:DB10_HMI_in/4:intensity/4:[23]
  ChannelDirection23 = OUT
  ChannelType23 = INT
  Channel24
  ChannelID24 = NIR2_Int24
  ChannelBrowsePath24 = /0:Root/0:Objects/3:ServerInterfaces/0:RecData/4:DB10_HMI_in/4:intensity/4:[24]
  ChannelDirection24 = OUT
  ChannelType24 = INT
  Channel25
  ChannelID25 = NIR2_Int25
  ChannelBrowsePath25 = /0:Root/0:Objects/3:ServerInterfaces/0:RecData/4:DB10_HMI_in/4:intensity/4:[25]
  ChannelDirection25 = OUT
  ChannelType25 = INT
  Channel26
  ChannelID26 = NIR2_Int26
  ChannelBrowsePath26 = /0:Root/0:Objects/3:ServerInterfaces/0:RecData/4:DB10_HMI_in/4:intensity/4:[26]
  ChannelDirection26 = OUT
  ChannelType26 = INT
  Channel27
  ChannelID27 = NIR2_Int27
  ChannelBrowsePath27 = /0:Root/0:Objects/3:ServerInterfaces/0:RecData/4:DB10_HMI_in/4:intensity/4:[27]
  ChannelDirection27 = OUT
  ChannelType27 = INT
  Channel28
  ChannelID28 = NIR2_Int28
  ChannelBrowsePath28 = /0:Root/0:Objects/3:ServerInterfaces/0:RecData/4:DB10_HMI_in/4:intensity/4:[28]
  ChannelDirection28 = OUT
  ChannelType28 = INT
  Channel29
  ChannelID29 = NIR2_Int29
  ChannelBrowsePath29 = /0:Root/0:Objects/3:ServerInterfaces/0:RecData/4:DB10_HMI_in/4:intensity/4:[29]
  ChannelDirection29 = OUT
  ChannelType29 = INT
  Channel30
  ChannelID30 = NIR2_Int30
  ChannelBrowsePath30 = /0:Root/0:Objects/3:ServerInterfaces/0:RecData/4:DB10_HMI_in/4:intensity/4:[30]
  ChannelDirection30 = OUT
  ChannelType30 = INT
  Channel31
  ChannelID31 = NIR2_Int31
  ChannelBrowsePath31 = /0:Root/0:Objects/3:ServerInterfaces/0:RecData/4:DB10_HMI_in/4:intensity/4:[31]
  ChannelDirection31 = OUT
  ChannelType31 = INT
  Channel32
  ChannelID32 = NIR2_Int32
  ChannelBrowsePath32 = /0:Root/0:Objects/3:ServerInterfaces/0:RecData/4:DB10_HMI_in/4:intensity/4:[32]
  ChannelDirection32 = OUT
  ChannelType32 = INT
  Channel33
  ChannelID33 = NIR2_Int33
  ChannelBrowsePath33 = /0:Root/0:Objects/3:ServerInterfaces/0:RecData/4:DB10_HMI_in/4:intensity/4:[33]
  ChannelDirection33 = OUT
  ChannelType33 = INT
  Channel34
  ChannelID34 = NIR2_Int34
  ChannelBrowsePath34 = /0:Root/0:Objects/3:ServerInterfaces/0:RecData/4:DB10_HMI_in/4:intensity/4:[34]
  ChannelDirection34 = OUT
  ChannelType34 = INT
  Channel35
  ChannelID35 = NIR2_Int35
  ChannelBrowsePath35 = /0:Root/0:Objects/3:ServerInterfaces/0:RecData/4:DB10_HMI_in/4:intensity/4:[35]
  ChannelDirection35 = OUT
  ChannelType35 = INT
  Channel36
  ChannelID36 = NIR2_Int36
  ChannelBrowsePath36 = /0:Root/0:Objects/3:ServerInterfaces/0:RecData/4:DB10_HMI_in/4:intensity/4:[36]
  ChannelDirection36 = OUT
  ChannelType36 = INT
  Channel37
  ChannelID37 = NIR2_Int37
  ChannelBrowsePath37 = /0:Root/0:Objects/3:ServerInterfaces/0:RecData/4:DB10_HMI_in/4:intensity/4:[37]
  ChannelDirection37 = OUT
  ChannelType37 = INT
  Channel38
  ChannelID38 = NIR2_Int38
  ChannelBrowsePath38 = /0:Root/0:Objects/3:ServerInterfaces/0:RecData/4:DB10_HMI_in/4:intensity/4:[38]
  ChannelDirection38 = OUT
  ChannelType38 = INT
  Channel39
  ChannelID39 = NIR2_Int39
  ChannelBrowsePath39 = /0:Root/0:Objects/3:ServerInterfaces/0:RecData/4:DB10_HMI_in/4:intensity/4:[39]
  ChannelDirection39 = OUT
  ChannelType39 = INT
  Channel40
  ChannelID40 = NIR2_Int40
  ChannelBrowsePath40 = /0:Root/0:Objects/3:ServerInterfaces/0:RecData/4:DB10_HMI_in/4:intensity/4:[40]
  ChannelDirection40 = OUT
  ChannelType40 = INT
  Channel41
  ChannelID41 = NIR2_Int41
  ChannelBrowsePath41 = /0:Root/0:Objects/3:ServerInterfaces/0:RecData/4:DB10_HMI_in/4:intensity/4:[41]
  ChannelDirection41 = OUT
  ChannelType41 = INT
  Channel42
  ChannelID42 = NIR2_Int42
  ChannelBrowsePath42 = /0:Root/0:Objects/3:ServerInterfaces/0:RecData/4:DB10_HMI_in/4:intensity/4:[42]
  ChannelDirection42 = OUT
  ChannelType42 = INT
  Channel43
  ChannelID43 = NIR2_Int43
  ChannelBrowsePath43 = /0:Root/0:Objects/3:ServerInterfaces/0:RecData/4:DB10_HMI_in/4:intensity/4:[43]
  ChannelDirection43 = OUT
  ChannelType43 = INT
  Channel44
  ChannelID44 = NIR2_Int44
  ChannelBrowsePath44 = /0:Root/0:Objects/3:ServerInterfaces/0:RecData/4:DB10_HMI_in/4:intensity/4:[44]
  ChannelDirection44 = OUT
  ChannelType44 = INT
  Channel45
  ChannelID45 = NIR2_Int45
  ChannelBrowsePath45 = /0:Root/0:Objects/3:ServerInterfaces/0:RecData/4:DB10_HMI_in/4:intensity/4:[45]
  ChannelDirection45 = OUT
  ChannelType45 = INT
  Channel46
  ChannelID46 = NIR2_Int46
  ChannelBrowsePath46 = /0:Root/0:Objects/3:ServerInterfaces/0:RecData/4:DB10_HMI_in/4:intensity/4:[46]
  ChannelDirection46 = OUT
  ChannelType46 = INT
  Channel47
  ChannelID47 = NIR2_Int47
  ChannelBrowsePath47 = /0:Root/0:Objects/3:ServerInterfaces/0:RecData/4:DB10_HMI_in/4:intensity/4:[47]
  ChannelDirection47 = OUT
  ChannelType47 = INT
  Channel48
  ChannelID48 = NIR2_Int48
  ChannelBrowsePath48 = /0:Root/0:Objects/3:ServerInterfaces/0:RecData/4:DB10_HMI_in/4:intensity/4:[48]
  ChannelDirection48 = OUT
  ChannelType48 = INT
Printer : OpcUa_any v1.0.0.1  [ETH1 -> NirAdphos2.ETH2 [Cable Type=PowerlinkCable, Length=10, Version=1.0.0.3]]
  ServerDiagnostics = on
  ServerEndpointUrl = opc.tcp://192.168.125.10:4840
  UserIdentifyToken = 1
  Username = PressCore
  Password = h98o76
  Channel1
  ChannelID1 = xRunTransport
  ChannelBrowsePath1 = /0:Root/0:Objects/4:PLC/4:Modules/6:&:&:/6:Global PV/6:gDryerRemoteData/6:Commands/6:xRunTransport
  Channel2
  ChannelID2 = xPrepareToDry
  ChannelBrowsePath2 = /0:Root/0:Objects/4:PLC/4:Modules/6:&:&:/6:Global PV/6:gDryerRemoteData/6:Commands/6:xPrepareToDry
  ChannelSamplingInterval2 = 200
  ChannelPublishingInterval2 = 400
  Channel3
  ChannelID3 = xStartDrying
  ChannelBrowsePath3 = /0:Root/0:Objects/4:PLC/4:Modules/6:&:&:/6:Global PV/6:gDryerRemoteData/6:Commands/6:xStartDrying
  ChannelSamplingInterval3 = 200
  ChannelPublishingInterval3 = 400
  Channel4
  ChannelID4 = xEnableNir
  ChannelBrowsePath4 = /0:Root/0:Objects/4:PLC/4:Modules/6:&:&:/6:Global PV/6:gDryerRemoteData/6:Parameters/6:xEnableNir
  ChannelSamplingInterval4 = 200
  ChannelPublishingInterval4 = 400
  Channel5
  ChannelID5 = xEnableArcLampDrying
  ChannelBrowsePath5 = /0:Root/0:Objects/4:PLC/4:Modules/6:&:&:/6:Global PV/6:gDryerRemoteData/6:Parameters/6:xEnableArcLamp
  ChannelSamplingInterval5 = 200
  ChannelPublishingInterval5 = 400
  Channel6
  ChannelID6 = rBeltSpeedSetPoint
  ChannelBrowsePath6 = /0:Root/0:Objects/4:PLC/4:Modules/6:&:&:/6:Global PV/6:gDryerRemoteData/6:Parameters/6:rBeltSpeedSetPoint
  ChannelType6 = REAL
  Channel7
  ChannelID7 = rBoardLength
  ChannelBrowsePath7 = /0:Root/0:Objects/4:PLC/4:Modules/6:&:&:/6:Global PV/6:gDryerRemoteData/6:Parameters/6:Media/6:rLength
  ChannelSamplingInterval7 = 200
  ChannelPublishingInterval7 = 400
  ChannelType7 = REAL
  Channel8
  ChannelID8 = rBoardWidth
  ChannelBrowsePath8 = /0:Root/0:Objects/4:PLC/4:Modules/6:&:&:/6:Global PV/6:gDryerRemoteData/6:Parameters/6:Media/6:rWidth
  ChannelSamplingInterval8 = 200
  ChannelPublishingInterval8 = 400
  ChannelType8 = REAL
  Channel9
  ChannelID9 = rBoardThickness
  ChannelBrowsePath9 = /0:Root/0:Objects/4:PLC/4:Modules/6:&:&:/6:Global PV/6:gDryerRemoteData/6:Parameters/6:Media/6:rThickness
  ChannelSamplingInterval9 = 200
  ChannelPublishingInterval9 = 400
  ChannelType9 = REAL
  Channel10
  ChannelID10 = rBoardGap
  ChannelBrowsePath10 = /0:Root/0:Objects/4:PLC/4:Modules/6:&:&:/6:Global PV/6:gDryerRemoteData/6:Parameters/6:Media/6:rGap
  ChannelSamplingInterval10 = 200
  ChannelPublishingInterval10 = 400
  ChannelType10 = REAL
  Channel11
  ChannelID11 = Signals_xMediaPresent
  ChannelBrowsePath11 = /0:Root/0:Objects/4:PLC/4:Modules/6:&:&:/6:Global PV/6:gDryerRemoteData/6:Signals/6:xMediaPresent
  ChannelSamplingInterval11 = 200
  ChannelPublishingInterval11 = 400
  Channel12
  ChannelID12 = Signals_xBreakerOKBlowerInput
  ChannelBrowsePath12 = /0:Root/0:Objects/4:PLC/4:Modules/6:&:&:/6:Global PV/6:gDryerRemoteData/6:Signals/6:xBreakerOKBlowerInput
  ChannelSamplingInterval12 = 200
  ChannelPublishingInterval12 = 400
  Channel13
  ChannelID13 = Signals_xBreakerOKBlowerOutput
  ChannelBrowsePath13 = /0:Root/0:Objects/4:PLC/4:Modules/6:&:&:/6:Global PV/6:gDryerRemoteData/6:Signals/6:xBreakerOKBlowerOutput
  ChannelSamplingInterval13 = 200
  ChannelPublishingInterval13 = 400
  Channel14
  ChannelID14 = Signals_Safety_xMovementsEnabled
  ChannelBrowsePath14 = /0:Root/0:Objects/4:PLC/4:Modules/6:&:&:/6:Global PV/6:gDryerRemoteData/6:Signals/6:Safety/6:xMovementsEnabled
  ChannelSamplingInterval14 = 200
  ChannelPublishingInterval14 = 400
  Channel15
  ChannelID15 = Signals_Safety_xRemoteEStopOK
  ChannelBrowsePath15 = /0:Root/0:Objects/4:PLC/4:Modules/6:&:&:/6:Global PV/6:gDryerRemoteData/6:Signals/6:Safety/6:xRemoteEStopOK
  ChannelSamplingInterval15 = 200
  ChannelPublishingInterval15 = 400
  Channel16
  ChannelID16 = Signals_Safety_xEStopFrontOK
  ChannelBrowsePath16 = /0:Root/0:Objects/4:PLC/4:Modules/6:&:&:/6:Global PV/6:gDryerRemoteData/6:Signals/6:Safety/6:xEStopFrontOK
  ChannelSamplingInterval16 = 200
  ChannelPublishingInterval16 = 400
  Channel17
  ChannelID17 = Signals_Safety_xEStopRearOK
  ChannelBrowsePath17 = /0:Root/0:Objects/4:PLC/4:Modules/6:&:&:/6:Global PV/6:gDryerRemoteData/6:Signals/6:Safety/6:xEStopRearOK
  ChannelSamplingInterval17 = 200
  ChannelPublishingInterval17 = 400
  Channel18
  ChannelID18 = Signals_Safety_xClosedFrontIn
  ChannelBrowsePath18 = /0:Root/0:Objects/4:PLC/4:Modules/6:&:&:/6:Global PV/6:gDryerRemoteData/6:Signals/6:Safety/6:xClosedFrontInput
  ChannelSamplingInterval18 = 200
  ChannelPublishingInterval18 = 400
  Channel19
  ChannelID19 = Signals_Safety_xClosedFrontOut
  ChannelBrowsePath19 = /0:Root/0:Objects/4:PLC/4:Modules/6:&:&:/6:Global PV/6:gDryerRemoteData/6:Signals/6:Safety/6:xClosedFrontOutput
  ChannelSamplingInterval19 = 200
  ChannelPublishingInterval19 = 400
  Channel20
  ChannelID20 = Signals_Safety_xClosedRearIn
  ChannelBrowsePath20 = /0:Root/0:Objects/4:PLC/4:Modules/6:&:&:/6:Global PV/6:gDryerRemoteData/6:Signals/6:Safety/6:xClosedRearInput
  ChannelSamplingInterval20 = 200
  ChannelPublishingInterval20 = 400
  Channel21
  ChannelID21 = Signals_Safety_xClosedRearOut
  ChannelBrowsePath21 = /0:Root/0:Objects/4:PLC/4:Modules/6:&:&:/6:Global PV/6:gDryerRemoteData/6:Signals/6:Safety/6:xClosedRearOutput
  ChannelSamplingInterval21 = 200
  ChannelPublishingInterval21 = 400
  Channel22
  ChannelID22 = rDocumentWidth
  ChannelBrowsePath22 = /0:Root/0:Objects/4:PLC/4:Modules/6:&:&:/6:Global PV/6:gDryerRemoteData/6:Parameters/6:Media/6:rDocWidth
  ChannelSamplingInterval22 = 200
  ChannelPublishingInterval22 = 400
  ChannelType22 = REAL
  Channel23
  ChannelID23 = rDocumentLength
  ChannelBrowsePath23 = /0:Root/0:Objects/4:PLC/4:Modules/6:&:&:/6:Global PV/6:gDryerRemoteData/6:Parameters/6:Media/6:rDocLength
  ChannelSamplingInterval23 = 200
  ChannelPublishingInterval23 = 400
  ChannelType23 = REAL
  Channel24
  ChannelID24 = xLineEmptyingBelt
  ChannelBrowsePath24 = /0:Root/0:Objects/4:PLC/4:Modules/6:&:&:/6:Global PV/6:gDryerRemoteData/6:Parameters/6:xLineEmptyingBelt
  ChannelSamplingInterval24 = 200
  ChannelPublishingInterval24 = 400
  Channel25
  ChannelID25 = xPrepareToEmptyBelt
  ChannelBrowsePath25 = /0:Root/0:Objects/4:PLC/4:Modules/6:&:&:/6:Global PV/6:gDryerRemoteData/6:Commands/6:xPrepareToEmptyBelt
  ChannelSamplingInterval25 = 200
  ChannelPublishingInterval25 = 400
  Channel26
  ChannelID26 = rDocumentOffset
  ChannelBrowsePath26 = /0:Root/0:Objects/4:PLC/4:Modules/6:&:&:/6:Global PV/6:gDryerRemoteData/6:Parameters/6:Media/6:rDocCrossOffset
  ChannelSamplingInterval26 = 200
  ChannelPublishingInterval26 = 400
  ChannelType26 = REAL
  Channel27
  ChannelID27 = rCrossOffset
  ChannelBrowsePath27 = /0:Root/0:Objects/4:PLC/4:Modules/6:&:&:/6:Global PV/6:gDryerRemoteData/6:Parameters/6:Media/6:rCrossOffset
  ChannelSamplingInterval27 = 200
  ChannelPublishingInterval27 = 400
  ChannelType27 = REAL
  Channel28
  ChannelID28 = rSubstratePowerReduction
  ChannelBrowsePath28 = /0:Root/0:Objects/4:PLC/4:Modules/6:&:&:/6:Global PV/6:gDryerRemoteData/6:Parameters/6:rSubstratePowerReduction
  ChannelSamplingInterval28 = 200
  ChannelPublishingInterval28 = 400
  ChannelType28 = REAL
  Channel29
  ChannelID29 = xEnableDDC
  ChannelBrowsePath29 = /0:Root/0:Objects/4:PLC/4:Modules/6:&:&:/6:Global PV/6:gDryerRemoteData/6:Parameters/6:xEnableDDC
  ChannelSamplingInterval29 = 200
  ChannelPublishingInterval29 = 400
  Channel30
  ChannelID30 = xPrinterBeltRuning
  ChannelBrowsePath30 = /0:Root/0:Objects/4:PLC/4:Modules/6:&:&:/6:Global PV/6:gDryerRemoteData/6:Parameters/6:xPrinterBeltRuning
  ChannelSamplingInterval30 = 200
  ChannelPublishingInterval30 = 400
X20AI8321_207 : X20AI8321 v1.5.0.0  [SS1 -> X20TB1F5.SS; SL -> X20BM11e.SL1]
  Supervision = off
  LowerLimit = -8192
  ChannelType01 = 4 to 20mA
  ChannelType02 = 4 to 20mA
  ChannelType03 = 4 to 20mA
  ChannelType04 = 4 to 20mA
  ChannelType05 = 4 to 20mA
  ChannelType06 = 4 to 20mA
  ChannelType07 = 4 to 20mA
  ChannelType08 = 4 to 20mA
X20AO4622_208 : X20AO4622 v1.3.0.0  [SS1 -> X20TB12b.SS; SL -> X20BM11f.SL1]
  Supervision = off
X20AT4222_209 : X20AT4222 v1.4.0.0  [SS1 -> X20TB12c.SS; SL -> X20BM11g.SL1]
  FunctionModel = FunctionModel001
  Supervision = off
  SensorType03 = off
  SensorType04 = off
X20BB57 : X20BB57 v1.2.0.0
  Connector IF7:
    Baudrate = 250000
    ActivateCanOpen = 1
    p100c_parametervalue = 1000
    p100d_parametervalue = 3
X20BM01 : X20BM01 v2.2.0.0  [X2X1 -> X20BM11b.X2X2]
X20BM11 : X20BM11 v1.1.0.0  [X2X1 -> X20BB57.IF6]
X20BM11a : X20BM11 v1.1.0.0  [X2X1 -> X20BM11.X2X2]
X20BM11b : X20BM11 v1.1.0.0  [X2X1 -> X20BM11a.X2X2]
X20BM11c : X20BM11 v1.1.0.0  [X2X1 -> X20BM01.X2X2]
X20BM11d : X20BM11 v1.1.0.0  [X2X1 -> X20BM11c.X2X2]
X20BM11e : X20BM11 v1.1.0.0  [X2X1 -> X20BM11d.X2X2]
X20BM11f : X20BM11 v1.1.0.0  [X2X1 -> X20BM11e.X2X2]
X20BM11g : X20BM11 v1.1.0.0  [X2X1 -> X20BM11f.X2X2]
X20CP0483 : X20CP0483 v1.6.0.0  [SL -> X20BB57.SL1]
  Connector IF2:
    ActivateDevice = 1
    HostName = efi_dryer
    Mode = Manual
    InternetAddress = 192.168.125.47
    SubnetMask = 255.255.255.0
    InaNodeNumber = 0
    ActivateSnmp = 2
  Connector IF3:
    DNAConfiguration = manual
    EplNatSubnet = 192.168.102.0
  ConfigurationID = Dryer
  UserPartitionSize = 0
  SimulationIPAddress = 192.168.0.138
  SimulationModeOpcUa = off
  PermanentPvSize = 5000
  RemanentGlobalPvSize = 10000
  VolatileGlobalPvSize = 1500000
  UserLoggerSize = 4096000
  EnableUsbRemoteInstall = 1
  EnableCfRemoteInstall = 1
  RebootReset = 1
  TimerDeviceType = EPLX2X
  TimerDevice = X20CP0483.IF3
  TaskClassIdleTime = 4000
  CyclicTaskClassCount = 6
  Cyclic1Duration = 8000
  Cyclic1Tolerance = 8000
  Cyclic1Stack = 16384
  Cyclic1Output = 1
  Cyclic2Duration = 12000
  Cyclic2Tolerance = 24000
  Cyclic2Stack = 16384
  Cyclic3Duration = 16000
  Cyclic3Tolerance = 48000
  Cyclic3Stack = 16384
  Cyclic4Duration = 32000
  Cyclic4Tolerance = 96000
  Cyclic4Stack = 16384
  Cyclic5Duration = 80000
  Cyclic5Tolerance = 160000
  Cyclic5Stack = 16384
  Cyclic6Duration = 88000
  Cyclic6Tolerance = 528000
  Cyclic7Duration = 1000000
  Cyclic7Tolerance = 1000000
  Cyclic8Duration = 800000
  Cyclic8Tolerance = 30400000
  FileDevice1
  FileDeviceName1 = USER
  FileDevicePath1 = USER_PATH
  FtpUser1
  FtpUsername1 = EFI  // EFI
  FtpUserPassword1 = 7G5n+wCoc8AAtJwOeMqQrBZ1Z+2KeIxeQkt+7Ofj72s=  // Castellon
  FtpUserSalt1 = xa1UK9Qk
  FTPAccessRight1 = 0
  FTPdevice1 = ALL
  ActivateOpcUa = 1
  OpcUaInformationModels_PV_Version = 2
  OpcUaInformationModel_Facet = 0
  OpcUaInformationModel_TypeInformation = 0
  OpcUaInformationModel_BaseObjectTypeForStructures = 0
X20DIF371_201 : X20DIF371 v1.3.0.0  [SS1 -> X20TB1F.SS; SL -> X20BM11.SL1]
  Supervision = off
X20DIF371_202 : X20DIF371 v1.3.0.0  [SS1 -> X20TB1F1.SS; SL -> X20BM11a.SL1]
  Supervision = off
X20DIF371_203 : X20DIF371 v1.3.0.0  [SS1 -> X20TB1F2.SS; SL -> X20BM11b.SL1]
  Supervision = off
X20DOF322_205 : X20DOF322 v1.5.0.0  [SS1 -> X20TB1F3.SS; SL -> X20BM11c.SL1]
  Supervision = off
X20DOF322_206 : X20DOF322 v1.5.0.0  [SS1 -> X20TB1F4.SS; SL -> X20BM11d.SL1]
  Supervision = off
X20PS3300_204 : X20PS3300 v1.4.0.0  [SS1 -> X20TB12a.SS; SL -> X20BM01.SL1]
  Supervision = off
X20PS9600 : X20PS9600 v1.6.0.0  [PS -> X20BB57.PS1; SS1 -> X20TB12.SS]
  Supervision = off
X20TB12 : X20TB12 v1.0.0.0
X20TB12a : X20TB12 v1.0.0.0
X20TB12b : X20TB12 v1.0.0.0
X20TB12c : X20TB12 v1.0.0.0
X20TB1F : X20TB1F v1.0.0.0
X20TB1F1 : X20TB1F v1.0.0.0
X20TB1F2 : X20TB1F v1.0.0.0
X20TB1F3 : X20TB1F v1.0.0.0
X20TB1F4 : X20TB1F v1.0.0.0
X20TB1F5 : X20TB1F v1.0.0.0
X20cHB2880 : X20cHB2880 v1.2.0.0  [ETH1 -> 24PortHub.ETH20 [Cable Type=PowerlinkCable, Length=10, Version=1.0.0.3]]
```

### Cpu.per - X20CP0483/Cpu.per
```iecst
VAR_CONFIG
	gPermanentVersion AT %M0; (* *)
	gPermanentSwBelt AT %M200; (* *)
	gPermanentSimpleBlock AT %M500; (* *)
	gPermanentTrVacuum AT %M1000; (* *)
	gPermanentNirAdphos AT %M1500; (* *)
	gPermanentArcLampGew AT %M2000; (* *)
	gPermanentDryer AT %M2500; (* *)
END_VAR
```

### Acp10cfg.ncc - X20CP0483/Motion/Acp10cfg.ncc
```
NcConfiguration (Version=5.12.2, NcSwId=Acp10)
  ACP10CF1_typ:
    cnt_nettrc_rec_drive = 1500
    bufsize_trace_upload = 1200
    tc_nc_man_task = Cyclic #2
    glob_pv_as_ncobject = Yes
    ncsys_dl_broadcast = Yes
    ncsys_dl_acp_reset = Yes
    safemc_log_err_to_ax = Yes
    network_init:
      ncsw_init_execute = Yes
      automatic_execute = Yes
      node_nr_warning = Yes
      net_err_before_ncact = Yes
    nettrc:
      enter_parsecrec = Yes
      enter_ncaction = Yes
      save_ring_startidx = Yes
    cam_prof_download:
      cam_dat_dl_parallel = No
      tc_cam_dl_parallel = Task class for NC Manager task
    plk_if[0]:
      if_name = IF3
      tc_CycDat_PLCopen = Task class for NC Manager task
      mc_broadcast_extdat = No
    sdc_if[0]:
      if_name = SDC_IF1
      mc_broadcast_size = 800
      mc_broadcast_extdat = No
```

## Configuration SimDryer

CPU , AutomationRuntime I4.93, Build 4.1.2

### Task classes (Cpu.sw)
```
Cyclic#2 (cycle 8000 us, tolerance 8000 us):
  BasicDetec <- ExtPack._Media.BasicDetectMediaCtrl.BasicDetectMediaCtrl_v1.BasicDetectMediaCtrl.prg
  ThickFast <- ExtPack._Media.ThicknessCtrl.ThicknessCtrl_v2.ThicknessCtrl_Fast.prg
Cyclic#3 (cycle 12000 us, tolerance 12000 us):
  InitAxis <- ExtPack._Motion.AxisCtrl.AxisCtrl_v2.InitAxisControl.prg
  Belt <- ExtPack._Motion.AxisCtrl.AxisCtrl_v2.AxisCtrl.prg
  BlockVert <- ExtPack._Motion.AxisCtrl.AxisCtrl_v2.AxisCtrl.prg
  InitInvert <- ExtPack._Motion.InverterCtrl.InverterCtrl_v1.InitInverterCtrl.prg
  InvCtrl_1 <- ExtPack._Motion.InverterCtrl.InverterCtrl_v1.InverterCtrl.prg
  InvCtrl_2 <- ExtPack._Motion.InverterCtrl.InverterCtrl_v1.InverterCtrl.prg
Cyclic#4 (cycle 32000 us, tolerance 32000 us):
  Initialize <- Dryer.Config.Initialize.prg
  SimDryer <- Dryer.Sim.SimDryer.prg
  PhysIn <- Dryer.PhysicalMapping.PhysicalMapInputs.prg
  ThickCtrl <- ExtPack._Media.ThicknessCtrl.ThicknessCtrl_v2.ThicknessCtrl.prg
  Dryer_Fast <- Dryer.DryerCtrl.DryerCtrl_Fast.prg
  BeltCtrl <- ExtPack._Transport.BeltCtrl.BeltCtrl_v1.BeltCtrl.prg
  InitSBlock <- ExtPack.SimpleBlockCtrl.SimpleBlockCtrl_v1.InitSimpleBlockCtrl.prg
  SBlock <- ExtPack.SimpleBlockCtrl.SimpleBlockCtrl_v1.SimpleBlockCtrl.prg
  InitTransV <- ExtPack._Transport.TransVacuumCtrl.TransVacuumCtrl_v1.InitTransVacuumCtrl.prg
  TransVac_1 <- ExtPack._Transport.TransVacuumCtrl.TransVacuumCtrl_v1.TransVacuumCtrl.prg
  ArcLampGew <- ExtPack._Cure.ArcLampGEW.ArcLampGew_v1.ArcLampGewCtrl.prg
  NIRAdphos <- ExtPack._Cure.NIRAdphos.NIRAdphos_v1.NIRAdphosCtrl.prg
  HMI <- Dryer.HMI.HMI.prg
  PhysOut <- Dryer.PhysicalMapping.PhysicalMapOutputs.prg
  InSBlockS <- ExtPack.SimpleBlockCtrl.SimpleBlockSim.SimpleBlockSim_v1.InitSimpleBlockSim.prg
  SBlockSim <- ExtPack.SimpleBlockCtrl.SimpleBlockSim.SimpleBlockSim_v1.SimpleBlockSim.prg
  ArcLampSim <- ExtPack._Cure.ArcLampGEW.ArcLampSim.ArcLampSim_v1.ArcLampSim.prg
  NirAdphSim <- ExtPack._Cure.NIRAdphos.NirAdphosSim.NirAdphosSim_v1.NirAdphosSim.prg
  InitTrVacS <- ExtPack._Transport.TransVacuumCtrl.TransVacuumSim.TransVacuumSim_v1.InitTransVacuumSim.prg
  TrVaccSim1 <- ExtPack._Transport.TransVacuumCtrl.TransVacuumSim.TransVacuumSim_v1.TransVacuumSim.prg
  InitJamDet <- ExtPack._Transport.JamDetectCtrl.JamDetect_v1.InitJamDetect.prg
  JamDetect <- ExtPack._Transport.JamDetectCtrl.JamDetect_v1.JamDetect.prg
  IniJamDetS <- ExtPack._Transport.JamDetectCtrl.JamDetectSim.JamDetectSim_v1.InitJamDetectSim.prg
  JamDetectS <- ExtPack._Transport.JamDetectCtrl.JamDetectSim.JamDetectSim_v1.JamDetectSim.prg
Cyclic#5 (cycle 80000 us, tolerance 80000 us):
  DryerConf <- Dryer.Config.MachineConfigurator.prg
  Dryer_Slow <- Dryer.DryerCtrl.DryerCtrl_Slow.prg
  EventLogGe <- ExtPack._Tools.EventLog.EventLog_v1.EventLogGen.prg
  SavePerman <- Dryer.Config.SavePermanent.prg
  SimUseReg <- ExtPack._Tools.SimUseRegister.SimUseRegister_1.SimUseRegister.prg
  ThickReadE <- ExtPack._Media.ThicknessCtrl.ThicknessCtrl_v2.ThickReadEnergy.prg
Cyclic#7 (cycle 44000 us, tolerance 88000 us):
  FunctionsT <- UnitTest.Tests.FunctionsTests.prg
  PrepDryer <- UnitTest.Dryer.PrepareDryer.prg
  BeltTests <- UnitTest.Dryer.BeltTests.prg
DataObjects: Acp10sys
NcDataObjects: AcpErrTxt <- AxisTables.AcpErrTxt.dob, acp10etxen <- AxisTables.acp10etxen.dob, BeltS1400a <- AxisTables.BeltS1400_a.dob, BeltS1400i <- AxisTables.BeltS1400_i.dob, BK1_i <- AxisTables.BK1_i.dob, BK_sim_a <- AxisTables.BK_sim_a.dob, BeltP4_i, BeltP4_a
Binaries: TCData, udbdef, arsvcreg, mvLoader, TCLang, OpcUaSrv, acp10cfg, Acp10map, iomap, asfw, arconfig, ashwd, sysconf, ashwac, Role, User, TC, gAlrHist, gAlrCore, EFIunits, EFIfunct, Config, OpcUaMap
Libraries: UnitTest, LibAssert1, UtWs, UtMgr, FBs, Functions, ConvertFun, runtime, brsystem, sys_lib, standard, AsSafety, FileIO, AsXml, astime, asstring, AsFifo, NcGlobal, AsBrStr, MTBasics, MTTypes, MTFilter, AsTCP, AsIecCon, AsIOAcc, AsBrMath, AsEPL, ArEventLog, Acp10_MC, Acp10par, Acp10sim, Acp10sdc, DataObj, EvLogLib, ArProject, AsHttp, BRSE_JSON, MpCom, MpAlarmX, MpBase, MpServer, AxisFunc, IecCheck, ThickLib, AsOpcUac, ErrACS380, powerlnk, aruser, arssl, assem, ascanopen, acp10man, asopcuas, asopcuac, vcresman, ashw, asarcfg
```

### Task classes (Cpu1.sw)
```

```

### Hardware
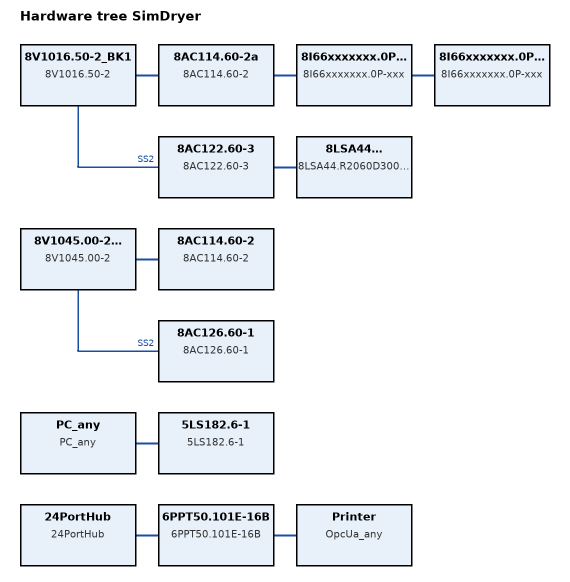
```
24PortHub : 24PortHub v1.0.0.1  [ETH1 -> 6PPT50.101E-16B.ETH1 [Cable Type=PowerlinkCable, Length=10, Version=1.0.0.3]; ETH12 -> PC_any.IF3 [Cable Type=PowerlinkCable, Length=10, Version=1.0.0.3]]
5LS182.6-1 : 5LS182.6-1 v1.5.0.0  [SL -> PC_any.SL1]
  Connector IF1:
    DNAConfiguration = manual
6PPT50.101E-16B : 6PPT50.101E-16B v1.3.8.0  [ETH1 -> 24PortHub.ETH1 [Cable Type=PowerlinkCable, Length=10, Version=1.0.0.3]; ETH2 -> Printer.ETH1 [Cable Type=PowerlinkCable, Length=10, Version=1.0.0.3]]
  Terminal = true
8AC114.60-2 : 8AC114.60-2 v1.0.0.8  [SS -> 8V1045.00-2_BELT.SS1; PLK1 -> 5LS182.6-1.IF1 [Cable Type=PowerlinkCable, Length=10, Version=1.0.0.3]; PLK2 -> 8AC114.60-2a.PLK1 [Cable Type=PowerlinkCable, Length=10, Version=1.0.0.3]]
8AC114.60-2a : 8AC114.60-2 v1.0.0.8  [SS -> 8V1016.50-2_BK1.SS1; PLK1 -> 8AC114.60-2.PLK2 [Cable Type=PowerlinkCable, Length=10, Version=1.0.0.3]; PLK2 -> 8I66xxxxxxx.0P-81.PLK1 [Cable Type=PowerlinkCable, Length=10, Version=1.0.0.3]]
8AC122.60-3 : 8AC122.60-3 v2.2.0.0  [SS -> 8V1016.50-2_BK1.SS2]
8AC126.60-1 : 8AC126.60-1 v2.2.0.0  [SS -> 8V1045.00-2_BELT.SS2]
8I66xxxxxxx.0P-81 : 8I66xxxxxxx.0P-xxx v2.5.1.0  [PLK1 -> 8AC114.60-2a.PLK2 (NodeNumber=81) [Cable Type=PowerlinkCable, Length=10, Version=1.0.0.3]; PLK2 -> 8I66xxxxxxx.0P-82.PLK1 (NodeNumber=81) [Cable Type=PowerlinkCable, Length=10, Version=1.0.0.3]]
  FunctionModel = Standard
  Supervision = off
  UnitOfSetpoint = Rpm
  Sel_AO1T = 0A
  Sel_NameplateMask = 8Ix6T401500_IEC
  Cfg_NSP = 2940
  Cfg_NCR = 277
  Cfg_COS = 82
  Sel_TUN = AUTO
8I66xxxxxxx.0P-82 : 8I66xxxxxxx.0P-xxx v2.5.1.0  [PLK1 -> 8I66xxxxxxx.0P-81.PLK2 [Cable Type=PowerlinkCable, Length=10, Version=1.0.0.3]]
  FunctionModel = Standard
  Supervision = off
  UnitOfSetpoint = Rpm
  Sel_AO1T = 0A
  Sel_NameplateMask = 8Ix6T401500_IEC
  Cfg_NSP = 2940
  Cfg_NCR = 277
  Cfg_COS = 82
  Sel_TUN = AUTO
8LSA44.R2060D300-3 : 8LSA44.R2060D300-3 v2.2.0.0  [EC -> 8AC122.60-3.EC; MT -> 8V1016.50-2_BK1.MT1]
8V1016.50-2_BK1 : 8V1016.50-2 v2.2.0.0
  MotionTP = Acp10Arnc0
8V1045.00-2_BELT : 8V1045.00-2 v2.2.0.0
  MotionTP = Acp10Arnc0
PC_any : PC_any v1.1.1.0 (OrderNumber=PC)
  Connector IF3:
    ActivateIna = 0
  ConfigurationID = SimDryer
  PermanentPvSize = 24000
  RemanentGlobalPvSize = 10000
  VolatileGlobalPvSize = 2000000
  SystemTick = 2000
  Cyclic1Duration = 4000
  Cyclic1Tolerance = 4000
  Cyclic1Stack = 32768
  Cyclic2Duration = 8000
  Cyclic2Tolerance = 8000
  Cyclic2Stack = 32768
  Cyclic3Duration = 12000
  Cyclic3Tolerance = 12000
  Cyclic3Stack = 32768
  Cyclic4Duration = 32000
  Cyclic4Tolerance = 32000
  Cyclic4Stack = 32768
  Cyclic5Duration = 80000
  Cyclic5Tolerance = 80000
  Cyclic5Stack = 32768
  Cyclic6Duration = 88000
  Cyclic6Tolerance = 88000
  Cyclic6Stack = 32768
  Cyclic7Duration = 44000
  Cyclic7Tolerance = 88000
  Cyclic7Stack = 32768
  Cyclic8Duration = 16000
  Cyclic8Tolerance = 16000
  Cyclic8Stack = 32768
  FileDevice1
  FileDeviceName1 = USER
  FileDevicePath1 = USER_PATH
  AnslPort = 11170
  FtpUser1
  FtpUsername1 = P4  // P4
  FtpUserPassword1 = LclxNYuP61nqo0LTZcDXp7yBDKZw4k3sO5UoQKFs6g8=  // efi
  FtpUserSalt1 = Ni00Nvek
  FTPAccessRight1 = 0
  WebServerPort = 83
  ActivateOpcUa = 1
  OpcUaPort = 4850
  OpcUaInformationModels_PV_Version = 2
  OpcUaInformationModel_Facet = 0
  OpcUaInformationModel_TypeInformation = 0
  OpcUaInformationModel_BaseObjectTypeForStructures = 0
Printer : OpcUa_any v1.0.0.1 (Disabled=true)  [ETH1 -> 6PPT50.101E-16B.ETH2 [Cable Type=PowerlinkCable, Length=10, Version=1.0.0.3]]
  Connector ETH2 (Disabled=true)
  ServerEndpointUrl = opc.tcp://192.168.125.10:4840
  Channel1
  ChannelID1 = xRunTransport
  ChannelBrowsePath1 = /0:Root/0:Objects/4:PLC/6:Modules/6:&:&:/6:Global PV/6:gDryerRemoteData/6:Commands/6:xRunTransport
  Channel2
  ChannelID2 = xPrepareToDry
  ChannelBrowsePath2 = /0:Root/0:Objects/4:PLC/6:Modules/6:&:&:/6:Global PV/6:gDryerRemoteData/6:Commands/6:xPrepareToDry
  Channel3
  ChannelID3 = xStartDrying
  ChannelBrowsePath3 = /0:Root/0:Objects/4:PLC/6:Modules/6:&:&:/6:Global PV/6:gDryerRemoteData/6:Commands/6:xStartDrying
  Channel4
  ChannelID4 = xEnableNirDrying
  ChannelBrowsePath4 = /0:Root/0:Objects/4:PLC/6:Modules/6:&:&:/6:Global PV/6:gDryerRemoteData/6:Commands/6:xEnableNirDrying
  Channel5
  ChannelID5 = xEnableArcLampDrying
  ChannelBrowsePath5 = /0:Root/0:Objects/4:PLC/6:Modules/6:&:&:/6:Global PV/6:gDryerRemoteData/6:Commands/6:xEnableArcLampDrying
  Channel6
  ChannelID6 = rBeltSpeedSetPoint
  ChannelBrowsePath6 = /0:Root/0:Objects/4:PLC/6:Modules/6:&:&:/6:Global PV/6:gDryerRemoteData/6:Parameters/6:rBeltSpeedSetPoint
  ChannelType6 = REAL
  Channel7
  ChannelID7 = rBoardLength
  ChannelBrowsePath7 = /0:Root/0:Objects/4:PLC/6:Modules/6:&:&:/6:Global PV/6:gDryerRemoteData/6:Parameters/6:Media/6:rLength
  ChannelType7 = REAL
  Channel8
  ChannelID8 = rBoardWidth
  ChannelBrowsePath8 = /0:Root/0:Objects/4:PLC/6:Modules/6:&:&:/6:Global PV/6:gDryerRemoteData/6:Parameters/6:Media/6:rWidth
  ChannelType8 = REAL
  Channel9
  ChannelID9 = rBoardThickness
  ChannelBrowsePath9 = /0:Root/0:Objects/4:PLC/6:Modules/6:&:&:/6:Global PV/6:gDryerRemoteData/6:Parameters/6:Media/6:rThickness
  ChannelType9 = REAL
  Channel10
  ChannelID10 = rBoardGap
  ChannelBrowsePath10 = /0:Root/0:Objects/4:PLC/6:Modules/6:&:&:/6:Global PV/6:gDryerRemoteData/6:Parameters/6:Media/6:rGap
  ChannelType10 = REAL
  Channel11
  ChannelID11 = Signals_xMediaPresent
  ChannelBrowsePath11 = /0:Root/0:Objects/4:PLC/6:Modules/6:&:&:/6:Global PV/6:gDryerRemoteData/6:Signals/6:xMediaPresent
  Channel12
  ChannelID12 = Signals_xBreakerOKBlowerInput
  ChannelBrowsePath12 = /0:Root/0:Objects/4:PLC/6:Modules/6:&:&:/6:Global PV/6:gDryerRemoteData/6:Signals/6:xBreakerOKBlowerInput
  Channel13
  ChannelID13 = Signals_xBreakerOKBlowerOutput
  ChannelBrowsePath13 = /0:Root/0:Objects/4:PLC/6:Modules/6:&:&:/6:Global PV/6:gDryerRemoteData/6:Signals/6:xBreakerOKBlowerOutput
  Channel14
  ChannelID14 = Signals_Safety_xMovementsEnabled
  ChannelBrowsePath14 = /0:Root/0:Objects/4:PLC/6:Modules/6:&:&:/6:Global PV/6:gDryerRemoteData/6:Signals/6:Safety/6:xMovementsEnabled
  Channel15
  ChannelID15 = Signals_Safety_xRemoteEStopOK
  ChannelBrowsePath15 = /0:Root/0:Objects/4:PLC/6:Modules/6:&:&:/6:Global PV/6:gDryerRemoteData/6:Signals/6:Safety/6:xRemoteEStopOK
  Channel16
  ChannelID16 = Signals_Safety_xEStopFrontOK
  ChannelBrowsePath16 = /0:Root/0:Objects/4:PLC/6:Modules/6:&:&:/6:Global PV/6:gDryerRemoteData/6:Signals/6:Safety/6:xEStopFrontOK
  Channel17
  ChannelID17 = Signals_Safety_xEStopRearOK
  ChannelBrowsePath17 = /0:Root/0:Objects/4:PLC/6:Modules/6:&:&:/6:Global PV/6:gDryerRemoteData/6:Signals/6:Safety/6:xEStopRearOK
  Channel18
  ChannelID18 = Signals_Safety_xClosedFrontIn
  ChannelBrowsePath18 = /0:Root/0:Objects/4:PLC/6:Modules/6:&:&:/6:Global PV/6:gDryerRemoteData/6:Signals/6:Safety/6:xClosedFrontInput
  Channel19
  ChannelID19 = Signals_Safety_xClosedFrontOut
  ChannelBrowsePath19 = /0:Root/0:Objects/4:PLC/6:Modules/6:&:&:/6:Global PV/6:gDryerRemoteData/6:Signals/6:Safety/6:xClosedFrontOutput
  Channel20
  ChannelID20 = Signals_Safety_xClosedRearIn
  ChannelBrowsePath20 = /0:Root/0:Objects/4:PLC/6:Modules/6:&:&:/6:Global PV/6:gDryerRemoteData/6:Signals/6:Safety/6:xClosedRearInput
  Channel21
  ChannelID21 = Signals_Safety_xClosedRearOut
  ChannelBrowsePath21 = /0:Root/0:Objects/4:PLC/6:Modules/6:&:&:/6:Global PV/6:gDryerRemoteData/6:Signals/6:Safety/6:xClosedRearOutput
  Channel22
  ChannelID22 = rDocumentWidth
  ChannelBrowsePath22 = /0:Root/0:Objects/4:PLC/6:Modules/6:&:&:/6:Global PV/6:gDryerRemoteData/6:Parameters/6:Document/6:rWidth
  ChannelSamplingInterval22 = 200
  ChannelPublishingInterval22 = 400
  ChannelType22 = REAL
  Channel23
  ChannelID23 = rDocumentLength
  ChannelBrowsePath23 = /0:Root/0:Objects/4:PLC/6:Modules/6:&:&:/6:Global PV/6:gDryerRemoteData/6:Parameters/6:Document/6:rLength
  ChannelSamplingInterval23 = 200
  ChannelPublishingInterval23 = 400
  ChannelType23 = REAL
  Channel24
  ChannelID24 = xLineEmptyingBelt
  ChannelBrowsePath24 = /0:Root/0:Objects/4:PLC/6:Modules/6:&:&:/6:Global PV/6:gDryerRemoteData/6:Parameters/6:xLineEmptyingBelt
  ChannelSamplingInterval24 = 200
  ChannelPublishingInterval24 = 400
  Channel25
  ChannelID25 = xPrepareToEmptyBelt
  ChannelBrowsePath25 = /0:Root/0:Objects/4:PLC/4:Modules/6:&amp;:&amp;:/6:Global PV/6:gDryerRemoteData/6:Commands/6:xPrepareToEmptyBelt
  ChannelSamplingInterval25 = 200
  ChannelPublishingInterval25 = 400
  Channel26
  ChannelID26 = xPrinterBeltRuning
  ChannelBrowsePath26 = /0:Root/0:Objects/4:PLC/6:Modules/6:&:&:/6:Global PV/6:gDryerRemoteData/6:Parameters/6:xPrinterBeltRuning
  ChannelSamplingInterval26 = 200
  ChannelPublishingInterval26 = 400
```

### Cpu.per - PC_any/Cpu.per
```iecst
VAR_CONFIG
	gPermanentSN AT %M0; (*Serial Number of the machine*)
	gPermanentSwBelt AT %M200; (* *)
END_VAR
```

### IoMap.iom - PC_any/IoMap.iom
```iecst
(********************************************************************
 * COPYRIGHT -- Bernecker + Rainer
 ********************************************************************
 * File: IoMap.iom
 * Author: B+R
 ********************************************************************
 * IO mapping file
 ********************************************************************)
VAR_CONFIG
	::gInverterSignalsPowerLink[1].In.ModuleOk AT %IX."8I66xxxxxxx.0P-81".ModuleOk;
	::gInverterSignalsPowerLink[1].In.StatusWord AT %IW."8I66xxxxxxx.0P-81".ETAD_Input;
	::gInverterSignalsPowerLink[1].Out.ControlWord AT %QW."8I66xxxxxxx.0P-81".CMDD_Output;
	::gInverterSignalsPowerLink[1].Out.SetSpeed AT %QW."8I66xxxxxxx.0P-81".LFRD_Output;
	::gInverterSignalsPowerLink[2].In.ModuleOk AT %IX."8I66xxxxxxx.0P-82".ModuleOk;
	::gInverterSignalsPowerLink[2].In.StatusWord AT %IW."8I66xxxxxxx.0P-82".ETAD_Input;
	::gInverterSignalsPowerLink[2].Out.ControlWord AT %QW."8I66xxxxxxx.0P-82".CMDD_Output;
	::gInverterSignalsPowerLink[2].Out.SetSpeed AT %QW."8I66xxxxxxx.0P-82".LFRD_Output;
	::gDryerAnc.Inputs.xTransportMoving AT %IX."Printer".xRuningBelt;
	::gDryerAnc.Outputs.xRunTransport AT %QX."Printer".xRunTransport;
	::gDryerAnc.Outputs.xPrepareToDry AT %QX."Printer".xPrepareToDry;
	::gDryerAnc.Outputs.xStartDrying AT %QX."Printer".xStartDrying;
	::gDryerAnc.Inputs.xDrying AT %IX."Printer".xDrying;
	::gDryerAnc.Inputs.xReadyToDry AT %IX."Printer".xReadyToDry;
	::gDryerAnc.Inputs.xReadyToEmptyBelt AT %IX."Printer".xReadyToEmptyBelt;
	::gDryerAnc.Inputs.xJamDetection AT %IX."Printer".xJamDetection;
	::gDryerAnc.Inputs.xTransportMoving AT %IX."Printer".xTransportMoving;
	::gDryerAnc.Inputs.xInRemote AT %IX."Printer".xInRemote;
	::gDryerAnc.Parameters.rSpeedSetPoint AT %QD."Printer".rBeltSpeedSetPoint;
	::gDryerAnc.Parameters.rMediaLength AT %QD."Printer".rBoardLength;
	::gDryerAnc.Parameters.rMediaWidth AT %QD."Printer".rBoardWidth;
	::gDryerAnc.Parameters.rMediaThickness AT %QD."Printer".rBoardThickness;
	::gDryerAnc.Parameters.rMediaGap AT %QD."Printer".rBoardGap;
	::gDryerRemoteData.Signals.xMediaPresent AT %QX."Printer".Signals_xMediaPresent;
	::gDryerRemoteData.Signals.xBreakerOKBlowerInput AT %QX."Printer".Signals_xBreakerOKBlowerInput;
	::gDryerRemoteData.Signals.xBreakerOKBlowerOutput AT %QX."Printer".Signals_xBreakerOKBlowerOutput;
	::gDryerRemoteData.Signals.Safety.xMovementsEnabled AT %QX."Printer".Signals_Safety_xMovementsEnabled;
	::gDryerRemoteData.Signals.Safety.xRemoteEStopOK AT %QX."Printer".Signals_Safety_xRemoteEStopOK;
	::gDryerRemoteData.Signals.Safety.xEStopFrontOK AT %QX."Printer".Signals_Safety_xEStopFrontOK;
	::gDryerRemoteData.Signals.Safety.xEStopRearOK AT %QX."Printer".Signals_Safety_xEStopRearOK;
	::gDryerRemoteData.Signals.Safety.xClosedFrontInput AT %QX."Printer".Signals_Safety_xClosedFrontIn;
	::gDryerRemoteData.Signals.Safety.xClosedFrontOutput AT %QX."Printer".Signals_Safety_xClosedFrontOut;
	::gDryerRemoteData.Signals.Safety.xClosedRearInput AT %QX."Printer".Signals_Safety_xClosedRearIn;
	::gDryerRemoteData.Signals.Safety.xClosedRearOutput AT %QX."Printer".Signals_Safety_xClosedRearOut;
	::gDryerRemoteData.Signals.xMediaPresent AT %IX."Printer".Signals_xMediaPresent;
	::gDryerRemoteData.Signals.xBreakerOKBlowerInput AT %IX."Printer".Signals_xBreakerOKBlowerInput;
	::gDryerRemoteData.Signals.xBreakerOKBlowerOutput AT %IX."Printer".Signals_xBreakerOKBlowerOutput;
	::gDryerRemoteData.Signals.Safety.xMovementsEnabled AT %IX."Printer".Signals_Safety_xMovementsEnabled;
	::gDryerRemoteData.Signals.Safety.xRemoteEStopOK AT %IX."Printer".Signals_Safety_xRemoteEStopOK;
	::gDryerRemoteData.Signals.Safety.xEStopFrontOK AT %IX."Printer".Signals_Safety_xEStopFrontOK;
	::gDryerRemoteData.Signals.Safety.xEStopRearOK AT %IX."Printer".Signals_Safety_xEStopRearOK;
	::gDryerRemoteData.Signals.Safety.xClosedFrontInput AT %IX."Printer".Signals_Safety_xClosedFrontIn;
	::gDryerRemoteData.Signals.Safety.xClosedFrontOutput AT %IX."Printer".Signals_Safety_xClosedFrontOut;
	::gDryerRemoteData.Signals.Safety.xClosedRearInput AT %IX."Printer".Signals_Safety_xClosedRearIn;
	::gDryerRemoteData.Signals.Safety.xClosedRearOutput AT %IX."Printer".Signals_Safety_xClosedRearOut;
	::gDryerRemoteData.Commands.xRunTransport AT %IX."Printer".xRunTransport;
	::gDryerRemoteData.Commands.xPrepareToDry AT %IX."Printer".xPrepareToDry;
	::gDryerRemoteData.Commands.xStartDrying AT %IX."Printer".xStartDrying;
	::gDryerRemoteData.Commands.xPrepareToEmptyBelt AT %IX."Printer".xPrepareToEmptyBelt;
	::gDryerRemoteData.Parameters.rBeltSpeedSetPoint AT %ID."Printer".rBeltSpeedSetPoint;
	::gDryerRemoteData.Parameters.Media.rLength AT %ID."Printer".rBoardLength;
	::gDryerRemoteData.Parameters.Media.rWidth AT %ID."Printer".rBoardWidth;
	::gDryerRemoteData.Parameters.Media.rThickness AT %ID."Printer".rBoardThickness;
	::gDryerRemoteData.Parameters.xEnableNir AT %IX."Printer".xEnableNirDrying;
	::gDryerRemoteData.Parameters.xEnableArcLamp AT %IX."Printer".xEnableArcLampDrying;
	::gDryerRemoteData.xCommsOK AT %IX."Printer".ModuleOk;
	::gDryerRemoteData.Parameters.Media.rDocWidth AT %ID."Printer".rDocumentWidth; (*Insert your comment here...*)
	::gDryerRemoteData.Parameters.Media.rDocLength AT %ID."Printer".rDocumentLength; (*Insert your comment here...*)
	::gDryerRemoteData.Parameters.xLineEmptyingBelt AT %IX."Printer".xLineEmptyingBelt;
	::gDryerRemoteData.Parameters.xPrinterBeltRuning AT %IX."Printer".xPrinterBeltRuning;
END_VAR
```

### Acp10cfg.ncc - PC_any/Motion/Acp10cfg.ncc
```
NcConfiguration (Version=5.02.1, NcSwId=Acp10)
  ACP10CF1_typ:
    cnt_nettrc_rec_drive = 1500
    bufsize_trace_upload = 1200
    tc_nc_man_task = Cyclic #1
    glob_pv_as_ncobject = Yes
    ncsys_dl_broadcast = Yes
    ncsys_dl_acp_reset = Yes
    safemc_log_err_to_ax = Yes
    network_init:
      ncsw_init_execute = Yes
      automatic_execute = No
      node_nr_warning = Yes
      net_err_before_ncact = Yes
    nettrc:
      enter_parsecrec = Yes
      enter_ncaction = Yes
      save_ring_startidx = Yes
    cam_prof_download:
      cam_dat_dl_parallel = No
      tc_cam_dl_parallel = Task class for NC Manager task
    plk_if[0]:
      if_name = SL1.IF1
      tc_CycDat_PLCopen = Task class for NC Manager task
      mc_broadcast_extdat = No
    sdc_if[0]:
      if_name = SDC_IF1
      mc_broadcast_size = 800
      mc_broadcast_extdat = No
```

### Acp10map.ncm - PC_any/Motion/Acp10map.ncm
```
NcMapping (NcSwId=Acp10, DisabledNodesAreHidden=False)
  NcObject gAxis01 (ModuleId=8V1045.00-2_BELT, Type=ncAXIS, Channel=1, AcoposSimulation=Off, InitParameter=BeltS1400i, AcoposParameter=BeltS1400a, Disabled=FALSE, ModuleDisabled=FALSE)
  NcObject 8V1045.00-2_ncV_AXIS1 (ModuleId=8V1045.00-2_BELT, Type=ncV_AXIS, Channel=1, Disabled=TRUE, ModuleDisabled=FALSE)
  NcObject gAxis02 (ModuleId=8V1016.50-2_BK1, Type=ncAXIS, Channel=1, AcoposSimulation=Off, InitParameter=BK1_i, AcoposParameter=BK_sim_a, Disabled=FALSE, ModuleDisabled=FALSE)
  NcObject 8V1016.50-2_ncV_AXIS1 (ModuleId=8V1016.50-2_BK1, Type=ncV_AXIS, Channel=1, Disabled=TRUE, ModuleDisabled=FALSE)
```

### EFIfunct.unittranslations - PC_any/UnitSystem/EFIfunct.unittranslations
```
Element UnitaryPercentage (Type=UnitTranslations)
  InputUnit:
    Namespace = http://www.opcfoundation.org/UA/units/un/cefact
    UnitID = 4404786
  OutputUnit:
    Namespace = http://www.opcfoundation.org/UA/units/un/cefact
    UnitID = 20529
  Formula = m * Input + n
  Formula_RPN = m Input * n +
  Formula_INV = (Output - n) / m
  Formula_INV_RPN = Output n - m /
  Variables:
    Variable_1:
      VariableId = m
      ProcessVariable = 
      StaticValue = 100
    Variable_2:
      VariableId = n
      ProcessVariable = 
      StaticValue = 0.0
```
